x summary
==================
This test method tests ``assert.bitNumber.x.valueIsLessThan``
method of CNM_AssertionInterfaces library, 
it provides the possibility to handover test data via parameter 


.. <legal notes>

legal notes
=================
| SPDX-FileCopyrightText: © 2022 ekvip automation GmbH <info@ekvip.de>
| SPDX-License-Identifier: Apache-2.0
| For details check: Apache-2.0_

.. _Apache-2.0: https://www.apache.org/licenses/LICENSE-2.0

.. </legal notes>

parameters
==========

*)

METHOD testValueIsLessThan
VAR_INPUT
	(* for the test it's the parameter ``currentValue`` *)
	valueToTest	:__XWORD;
	(* for the test it's the parameter ``greaterValue`` *)
	greater		:__XWORD;
END_VAR
VAR
	(* just the expectation if the assertion to test must be worng or true *)
	assertionIsWrong		:BOOL;
	(* contains the format string for the test message *)
	message					:Tc2_System.T_MaxString;
	(* TwinCAT printf with the test message *)
	messageStringBuilder	:Tc2_Utilities.FB_FormatString;
END_VAR
THIS^.assertorContainer.resetAssertor();

assertionIsWrong := (valueToTest >= greater);
message := SEL(
	assertionIsWrong,
	'currentValue is %d greaterValue is %d assertion must be TRUE',
	'currentValue is %d greaterValue is %d assertion must be FALSE'
);
messageStringBuilder(
	sFormat := message,
	arg1 := THIS^.AnyToArg(valueToTest),
	arg2 := THIS^.AnyToArg(greater)
);

THIS^.assertorContainer.assertor.assert.bitNumber.x.valueIsLessThan(
	currentValue := valueToTest,
	greaterValue := greater,
	message := ''
);

THIS^.AssertEquals_BOOL(
	Expected 	:= assertionIsWrong,
	Actual 		:= THIS^.assertorContainer.wasAssertionWrong,
	Message 	:= messageStringBuilder.sOut
);
END_METHOD

(*

x summary
==================
This test method tests ``assert.bitNumber.x.valueIsMax``
method of CNM_AssertionInterfaces library, 
it provides the possibility to handover test data via parameter 


.. <legal notes>

legal notes
=================
| SPDX-FileCopyrightText: © 2022 ekvip automation GmbH <info@ekvip.de>
| SPDX-License-Identifier: Apache-2.0
| For details check: Apache-2.0_

.. _Apache-2.0: https://www.apache.org/licenses/LICENSE-2.0

.. </legal notes>

parameters
==========

*)

METHOD testValueIsMax 
VAR_INPUT
	(* for the test it's the parameter ``currentValue`` *)
	valueToTest	:__XWORD;
	(* for the test it's the parameter ``maximumValue`` *)
	maximum		:__XWORD;
END_VAR
VAR
	(* just the expectation if the assertion to test must be worng or true *)
	assertionIsWrong		:BOOL;
	(* contains the format string for the test message *)
	message					:Tc2_System.T_MaxString;
	(* TwinCAT printf with the test message *)
	messageStringBuilder	:Tc2_Utilities.FB_FormatString;
END_VAR
THIS^.assertorContainer.resetAssertor();

assertionIsWrong := (valueToTest > maximum);
message := SEL(
	assertionIsWrong,
	'currentValue is %d maximumValue is %d assertion must be TRUE',
	'currentValue is %d maximumValue is %d assertion must be FALSE'
);
messageStringBuilder(
	sFormat := message,
	arg1 := THIS^.AnyToArg(valueToTest),
	arg2 := THIS^.AnyToArg(maximum)
);

THIS^.assertorContainer.assertor.assert.bitNumber.x.valueIsMax(
	currentValue := valueToTest,
	maximumValue := maximum,
	message := ''
);

THIS^.AssertEquals_BOOL(
	Expected 	:= assertionIsWrong,
	Actual 		:= THIS^.assertorContainer.wasAssertionWrong,
	Message 	:= messageStringBuilder.sOut
);
END_METHOD

(*

x summary
==================
This test method tests ``assert.bitNumber.x.valueIsMin``
method of CNM_AssertionInterfaces library, 
it provides the possibility to handover test data via parameter 


.. <legal notes>

legal notes
=================
| SPDX-FileCopyrightText: © 2022 ekvip automation GmbH <info@ekvip.de>
| SPDX-License-Identifier: Apache-2.0
| For details check: Apache-2.0_

.. _Apache-2.0: https://www.apache.org/licenses/LICENSE-2.0

.. </legal notes>

parameters
==========

*)

METHOD testValueIsMin 
VAR_INPUT
	(* for the test it's the parameter ``currentValue`` *)
	valueToTest	:__XWORD;
	(* for the test it's the parameter ``minimumValue`` *)
	minimum		:__XWORD;
END_VAR
VAR
	(* just the expectation if the assertion to test must be worng or true *)
	assertionIsWrong		:BOOL;
	(* contains the format string for the test message *)
	message					:Tc2_System.T_MaxString;
	(* TwinCAT printf with the test message *)
	messageStringBuilder	:Tc2_Utilities.FB_FormatString;
END_VAR
THIS^.assertorContainer.resetAssertor();

assertionIsWrong := (valueToTest < minimum);
message := SEL(
	assertionIsWrong,
	'currentValue is %d minimumValue is %d assertion must be TRUE',
	'currentValue is %d minimumValue is %d assertion must be FALSE'
);
messageStringBuilder(
	sFormat := message,
	arg1 := THIS^.AnyToArg(valueToTest),
	arg2 := THIS^.AnyToArg(minimum)
);

THIS^.assertorContainer.assertor.assert.bitNumber.x.valueIsMin(
	currentValue := valueToTest,
	minimumValue := minimum,
	message := ''
);

THIS^.AssertEquals_BOOL(
	Expected 	:= assertionIsWrong,
	Actual 		:= THIS^.assertorContainer.wasAssertionWrong,
	Message 	:= messageStringBuilder.sOut
);
END_METHOD

(*

x summary
==================
This test method tests ``assert.bitNumber.x.valueIsNotEqualTo``
method of CNM_AssertionInterfaces library, 
it provides the possibility to handover test data via parameter 


.. <legal notes>

legal notes
=================
| SPDX-FileCopyrightText: © 2022 ekvip automation GmbH <info@ekvip.de>
| SPDX-License-Identifier: Apache-2.0
| For details check: Apache-2.0_

.. _Apache-2.0: https://www.apache.org/licenses/LICENSE-2.0

.. </legal notes>

parameters
==========

*)

METHOD testValueIsNotEqualTo
VAR_INPUT
	(* for the test it's the parameter ``currentValue`` *)
	valueToTest	:__XWORD;
	(* for the test it's the parameter ``unexpectedValue`` *)
	unexpected	:__XWORD;
END_VAR
VAR
	(* just the expectation if the assertion to test must be worng or true *)
	assertionIsWrong		:BOOL;
	(* contains the format string for the test message *)
	message					:Tc2_System.T_MaxString;
	(* TwinCAT printf with the test message *)
	messageStringBuilder	:Tc2_Utilities.FB_FormatString;
END_VAR
THIS^.assertorContainer.resetAssertor();

assertionIsWrong := (valueToTest = unexpected);
message := SEL(
	assertionIsWrong,
	'currentValue is %d unexpectedValue is %d assertion must be TRUE', 
	'currentValue is %d unexpectedValue is %d assertion must be FALSE'
);
messageStringBuilder(
	sFormat := message,
	arg1 := THIS^.AnyToArg(valueToTest),
	arg2 := THIS^.AnyToArg(unexpected)
);

THIS^.assertorContainer.assertor.assert.bitNumber.x.valueIsNotEqualTo(
	currentValue := valueToTest,
	unexpectedValue := unexpected,
	message := ''
);

THIS^.AssertEquals_BOOL(
	Expected 	:= assertionIsWrong,
	Actual 		:= THIS^.assertorContainer.wasAssertionWrong,
	Message 	:= messageStringBuilder.sOut
);
END_METHOD

(*

x summary
==================
This test method tests ``assert.bitNumber.x.xorMaskIsEqualTo``
method of CNM_AssertionInterfaces library, 
it provides the possibility to handover test data via parameter 


.. <legal notes>

legal notes
=================
| SPDX-FileCopyrightText: © 2022 ekvip automation GmbH <info@ekvip.de>
| SPDX-License-Identifier: Apache-2.0
| For details check: Apache-2.0_

.. _Apache-2.0: https://www.apache.org/licenses/LICENSE-2.0

.. </legal notes>

parameters
==========

*)

METHOD testXorMaskIsEqualTo 
VAR_INPUT
	(* for the test it's the parameter ``currentValue`` *)
	valueToTest	:__XWORD;
	(* it's the mask for the currentValue *)
	mask		:__XWORD;
	(* for the test it's the parameter ``expectedValue`` *)
	expected	:__XWORD;
END_VAR
VAR
	(* just the expectation if the assertion to test must be worng or true *)
	assertionIsWrong		:BOOL;
	(* result of the bit operation to determine the value of ``assertionIsWrong`` *)
	result					:__XWORD;
	(* contains the format string for the test message *)
	message					:Tc2_System.T_MaxString;
	(* TwinCAT printf with the test message *)
	messageStringBuilder	:Tc2_Utilities.FB_FormatString;
END_VAR
THIS^.assertorContainer.resetAssertor();

result := (valueToTest XOR mask);
assertionIsWrong := (result <> expected);
message := SEL(
	assertionIsWrong,
	'currentValue: 16#%.16X XOR mask: 16#%.16X is 16#%.16X expectedValue: 16#%.16X assertion must be TRUE', 
	'currentValue: 16#%.16X XOR mask: 16#%.16X is 16#%.16X expectedValue: 16#%.16X assertion must be FALSE'
);
messageStringBuilder(
	sFormat := message,
	arg1 := THIS^.AnyToArg(valueToTest),
	arg2 := THIS^.AnyToArg(mask),
	arg3 := THIS^.AnyToArg(result),
	arg4 := THIS^.AnyToArg(expected)
);

THIS^.assertorContainer.assertor.assert.bitNumber.x.xorMaskIsEqualTo(
	currentValue	:= valueToTest,
	mask 			:= mask,
	expectedValue	:= expected,
	message			:= ''
);

THIS^.AssertEquals_BOOL(
	Expected 	:= assertionIsWrong,
	Actual 		:= THIS^.assertorContainer.wasAssertionWrong,
	Message 	:= messageStringBuilder.sOut
);
END_METHOD

(*

x summary
==================
This test method tests ``assert.bitNumber.x.xorMaskIsNotEqualTo``
method of CNM_AssertionInterfaces library, 
it provides the possibility to handover test data via parameter 


.. <legal notes>

legal notes
=================
| SPDX-FileCopyrightText: © 2022 ekvip automation GmbH <info@ekvip.de>
| SPDX-License-Identifier: Apache-2.0
| For details check: Apache-2.0_

.. _Apache-2.0: https://www.apache.org/licenses/LICENSE-2.0

.. </legal notes>

parameters
==========

*)

METHOD testXorMaskIsNotEqualTo 
VAR_INPUT
	(* for the test it's the parameter ``currentValue`` *)
	valueToTest	:__XWORD;
	(* it's the mask for the currentValue *)
	mask		:__XWORD;
	(* for the test it's the parameter ``unexpectedValue`` *)
	unexpected	:__XWORD;
END_VAR
VAR
	(* just the expectation if the assertion to test must be worng or true *)
	assertionIsWrong		:BOOL;
	(* result of the bit operation to determine the value of ``assertionIsWrong`` *)
	result					:__XWORD;
	(* contains the format string for the test message *)
	message					:Tc2_System.T_MaxString;
	(* TwinCAT printf with the test message *)
	messageStringBuilder	:Tc2_Utilities.FB_FormatString;
END_VAR
THIS^.assertorContainer.resetAssertor();

result := (valueToTest XOR mask);
assertionIsWrong := (result = unexpected);
message := SEL(
	assertionIsWrong,
	'currentValue: 16#%.16X XOR mask: 16#%.16X is 16#%.16X unexpectedValue: 16#%.16X assertion must be TRUE', 
	'currentValue: 16#%.16X XOR mask: 16#%.16X is 16#%.16X unexpectedValue: 16#%.16X assertion must be FALSE'
);
messageStringBuilder(
	sFormat := message,
	arg1 := THIS^.AnyToArg(valueToTest),
	arg2 := THIS^.AnyToArg(mask),
	arg3 := THIS^.AnyToArg(result),
	arg4 := THIS^.AnyToArg(unexpected)
);

THIS^.assertorContainer.assertor.assert.bitNumber.x.xorMaskIsNotEqualTo(
	currentValue	:= valueToTest,
	mask 			:= mask,
	unexpectedValue	:= unexpected,
	message			:= ''
);

THIS^.AssertEquals_BOOL(
	Expected 	:= assertionIsWrong,
	Actual 		:= THIS^.assertorContainer.wasAssertionWrong,
	Message 	:= messageStringBuilder.sOut
);
END_METHOD

END_FUNCTION_BLOCK

// ---- AssertionTester/AssertionTests/BitNumberAssertions/classes/LWordAssertionTests.TcPOU
(*

long summary
==================
This class tests all methods of LWORD assertions
with various combinations of inputs and checks expected 
outputs are satisfied or not

.. <legal notes>

legal notes
=================
| SPDX-FileCopyrightText: © 2022 ekvip automation GmbH <info@ekvip.de>
| SPDX-License-Identifier: Apache-2.0
| For details check: Apache-2.0_

.. _Apache-2.0: https://www.apache.org/licenses/LICENSE-2.0

.. </legal notes>

methods and properties
======================

*)

FUNCTION_BLOCK LWordAssertionTests EXTENDS AbstractAssertorTest
VAR_INPUT
END_VAR
VAR CONSTANT
	(* number of the lsb *)
	FIRST_BIT				:USINT := 0;
	(* number of the msb *)
	LAST_BIT				:USINT := 63;
	(* just the value zero *)
	ZERO					:LINT := 0;
	(* no single bit is set, it's just the value zero *)
	NO_BIT_SET				:LWORD := 16#0000_0000_0000_0000;
	(* just the lsb is set, it's just the value one *)
	LSB_ONLY				:LWORD := 16#0000_0000_0000_0001;
	(* all bits are set *)
	ALL_BITS_SET			:LWORD := 16#FFFF_FFFF_FFFF_FFFF;
	(* the msb is set only *)
	MSB_ONLY				:LWORD := 16#8000_0000_0000_0000;
	(* prefix to unify the test names *)
	TEST_NAME_PREFIX		:STRING := 'assert.bitNumber.long.';
	(* number how many times the product will be rotated right *)
	NUMBER_OF_RORS			:ULINT := 1;
	(* multiplicand for the ``multiplier`` *)
	MULTIPLICAND			:ULINT := 16#1111_1111_1111_1111;
	(* first of all multipliers the test iterates *)
	FIRST_MULTIPLIER		:ULINT := 0;
	(* first of all multipliers the test iterates *)
	LAST_MULTIPLIER			:ULINT := 15;
	(* constant for the modulo operator to check if valueToTest is even (lsb is unset) or odd (lsb is set) *)
	DEVISOR_FOR_EVEN_ODD	:ULINT := 2;
END_VAR

THIS^.runAndMaskIsEqualToTests();
THIS^.runAndMaskIsNotEqualToTests();
THIS^.runBitXIsEqualToTests();
THIS^.runBitXIsNotEqualToTests();
THIS^.runBitXIsSetTests();
THIS^.runBitXIsUnsetTests();
THIS^.runLsbIsEqualToTests();
THIS^.runLsbIsNotEqualToTests();
THIS^.runLsbIsSetTests();
THIS^.runLsbIsUnsetTests();
THIS^.runMsbIsEqualToTests();
THIS^.runMsbIsNotEqualToTests();
THIS^.runMsbIsSetTests();
THIS^.runMsbIsUnsetTests();
THIS^.runOrMaskIsEqualToTests();
THIS^.runOrMaskIsNotEqualToTests();
THIS^.runValueIsMaxTests();
THIS^.runValueIsMinTests();
THIS^.runValueIsEqualToTests();
THIS^.runValueIsGreaterTests();
THIS^.runValueIsLessThanTests();
THIS^.runValueIsInRangeOfTests();
THIS^.runValueIsNotEqualToTests();
THIS^.runXorMaskIsEqualToTests();
THIS^.runXorMaskIsNotEqualToTests();

(*

long summary
==================
This test method is a helper function to create a unified test name

.. <legal notes>

legal notes
=================
| SPDX-FileCopyrightText: © 2022 ekvip automation GmbH <info@ekvip.de>
| SPDX-License-Identifier: Apache-2.0
| For details check: Apache-2.0_

.. _Apache-2.0: https://www.apache.org/licenses/LICENSE-2.0

.. </legal notes>

parameters
==========

*)

METHOD PROTECTED getTestNameFor :Tc2_System.T_MaxString
VAR_INPUT
	(* name of the method to test, to create a unified test name *)
	nameOfMethodToTest	:Tc2_System.T_MaxString;
END_VAR
getTestNameFor := Tc2_Standard.CONCAT(THIS^.TEST_NAME_PREFIX, nameOfMethodToTest);
END_METHOD

(*

long summary
==================
This test method tests ``assert.bitNumber.long.andMaskIsEqualTo``
method of CNM_AssertionInterfaces library with various inputs

.. <legal notes>

legal notes
=================
| SPDX-FileCopyrightText: © 2022 ekvip automation GmbH <info@ekvip.de>
| SPDX-License-Identifier: Apache-2.0
| For details check: Apache-2.0_

.. _Apache-2.0: https://www.apache.org/licenses/LICENSE-2.0

.. </legal notes>

*)

METHOD runAndMaskIsEqualToTests
VAR
	(* shift to iterate through the bit numbers *)
	shift				:ULINT;
	(* mask with the bit iteration *)
	mask				:LWORD;
END_VAR
RETURN (NOT TcUnit.TEST_ORDERED(THIS^.getTestNameFor('AndMaskIsEqualTo')));

FOR shift:= THIS^.FIRST_BIT TO THIS^.LAST_BIT DO
	mask := SHL(THIS^.LSB_ONLY, shift);
	THIS^.testAndMaskIsEqualTo(
		valueToTest := THIS^.ALL_BITS_SET,
		mask  := mask,
		expected := mask
	);
	THIS^.testAndMaskIsEqualTo(
		valueToTest := THIS^.ALL_BITS_SET,
		mask  := mask,
		expected := (NOT mask)
	);
	THIS^.testAndMaskIsEqualTo(
		valueToTest := mask,
		mask  := (NOT mask),
		expected := THIS^.NO_BIT_SET
	);
	THIS^.testAndMaskIsEqualTo(
		valueToTest := mask,
		mask  := (NOT mask),
		expected := (NOT mask)
	);	
	THIS^.testAndMaskIsEqualTo(
		valueToTest := mask,
		mask  := mask,
		expected := mask
	);	
END_FOR

THIS^.testAndMaskIsEqualTo(
	valueToTest := THIS^.NO_BIT_SET,
	mask  := THIS^.NO_BIT_SET,
	expected := THIS^.NO_BIT_SET
);
THIS^.testAndMaskIsEqualTo(
	valueToTest := THIS^.NO_BIT_SET,
	mask  := THIS^.NO_BIT_SET,
	expected := THIS^.LSB_ONLY
);

THIS^.testAndMaskIsEqualTo(
	valueToTest := THIS^.ALL_BITS_SET,
	mask  := THIS^.ALL_BITS_SET,
	expected := THIS^.ALL_BITS_SET
);
THIS^.testAndMaskIsEqualTo(
	valueToTest := THIS^.ALL_BITS_SET,
	mask  := THIS^.ALL_BITS_SET,
	expected := THIS^.NO_BIT_SET
);

TcUnit.TEST_FINISHED();
END_METHOD

(*

long summary
==================
This test method tests ``assert.bitNumber.long.andMaskIsNotEqualTo``
method of CNM_AssertionInterfaces library with various inputs

.. <legal notes>

legal notes
=================
| SPDX-FileCopyrightText: © 2022 ekvip automation GmbH <info@ekvip.de>
| SPDX-License-Identifier: Apache-2.0
| For details check: Apache-2.0_

.. _Apache-2.0: https://www.apache.org/licenses/LICENSE-2.0

.. </legal notes>

*)

METHOD runAndMaskIsNotEqualToTests
VAR
	(* shift to iterate through the bit numbers *)
	shift	:ULINT;
	(* mask with the bit iteration *)
	mask	:LWORD;
END_VAR
RETURN (NOT TcUnit.TEST_ORDERED(THIS^.getTestNameFor('AndMaskIsNotEqualTo')));

FOR shift:= THIS^.FIRST_BIT TO THIS^.LAST_BIT DO
	mask := SHL(THIS^.LSB_ONLY, shift);
	THIS^.testAndMaskIsNotEqualTo(
		valueToTest := THIS^.ALL_BITS_SET,
		mask  := mask,
		unexpected := (NOT mask)
	);
	THIS^.testAndMaskIsNotEqualTo(
		valueToTest := THIS^.ALL_BITS_SET,
		mask  := mask,
		unexpected := mask
	);
	THIS^.testAndMaskIsNotEqualTo(
		valueToTest := mask,
		mask  := (NOT mask),
		unexpected := (NOT mask)
	);	
	THIS^.testAndMaskIsNotEqualTo(
		valueToTest := mask,
		mask  := (NOT mask),
		unexpected := THIS^.NO_BIT_SET
	);
	THIS^.testAndMaskIsNotEqualTo(
		valueToTest := mask,
		mask  := mask,
		unexpected := mask
	);	
END_FOR

THIS^.testAndMaskIsNotEqualTo(
	valueToTest := THIS^.NO_BIT_SET,
	mask  := THIS^.NO_BIT_SET,
	unexpected := THIS^.LSB_ONLY
);
THIS^.testAndMaskIsNotEqualTo(
	valueToTest := THIS^.NO_BIT_SET,
	mask  := THIS^.NO_BIT_SET,
	unexpected := THIS^.NO_BIT_SET
);

THIS^.testAndMaskIsNotEqualTo(
	valueToTest := THIS^.ALL_BITS_SET,
	mask  := THIS^.ALL_BITS_SET,
	unexpected := THIS^.NO_BIT_SET
);
THIS^.testAndMaskIsNotEqualTo(
	valueToTest := THIS^.ALL_BITS_SET,
	mask  := THIS^.ALL_BITS_SET,
	unexpected := THIS^.ALL_BITS_SET
);

TcUnit.TEST_FINISHED();
END_METHOD

(*

long summary
==================
This test method tests ``assert.bitNumber.long.bitXIsEqualTo``
method of CNM_AssertionInterfaces library with various inputs

.. <legal notes>

legal notes
=================
| SPDX-FileCopyrightText: © 2022 ekvip automation GmbH <info@ekvip.de>
| SPDX-License-Identifier: Apache-2.0
| For details check: Apache-2.0_

.. _Apache-2.0: https://www.apache.org/licenses/LICENSE-2.0

.. </legal notes>

*)

METHOD runBitXIsEqualToTests
VAR
	(* this is the number of the bit to test *)
	bitNumberToTest	:CNM_AssertionInterfaces.BitNumberLWord;
	(* it's just part of the test data *)
	valueToTest		:LWORD;
END_VAR
RETURN (NOT TcUnit.TEST_ORDERED(THIS^.getTestNameFor('bitXIsEqualTo')));

FOR bitNumberToTest := THIS^.FIRST_BIT TO THIS^.LAST_BIT DO

	valueToTest := SHL(THIS^.LSB_ONLY,bitNumberToTest);
	THIS^.testBitXIsEqualTo(
		valueToTest			:=valueToTest,
		bitNumberToCheck	:=bitNumberToTest,
		bitIsSet			:=TRUE
	);
	THIS^.testBitXIsEqualTo(
		valueToTest			:=valueToTest,
		bitNumberToCheck	:=bitNumberToTest,
		bitIsSet			:=FALSE
	);

	valueToTest := (NOT valueToTest);
	THIS^.testBitXIsEqualTo(
		valueToTest			:=valueToTest,
		bitNumberToCheck	:=bitNumberToTest,
		bitIsSet			:=FALSE
	);
	THIS^.testBitXIsEqualTo(
		valueToTest			:=valueToTest,
		bitNumberToCheck	:=bitNumberToTest,
		bitIsSet			:=TRUE
	);	
END_FOR

TcUnit.TEST_FINISHED();
END_METHOD

(*

long summary
==================
This test method tests ``assert.bitNumber.long.bitXIsNotEqualTo``
method of CNM_AssertionInterfaces library with various inputs

.. <legal notes>

legal notes
=================
| SPDX-FileCopyrightText: © 2022 ekvip automation GmbH <info@ekvip.de>
| SPDX-License-Identifier: Apache-2.0
| For details check: Apache-2.0_

.. _Apache-2.0: https://www.apache.org/licenses/LICENSE-2.0

.. </legal notes>

*)

METHOD runBitXIsNotEqualToTests
VAR
	(* this is the number of the bit to test *)
	bitNumberToTest	:CNM_AssertionInterfaces.BitNumberLWord;
	(* it's just part of the test data *)
	valueToTest		:LWORD;
END_VAR
RETURN (NOT TcUnit.TEST_ORDERED(THIS^.getTestNameFor('bitXIsNotEqualTo')));

FOR bitNumberToTest := THIS^.FIRST_BIT TO THIS^.LAST_BIT DO
	valueToTest := SHL(THIS^.LSB_ONLY,bitNumberToTest);
	THIS^.testBitXIsNotEqualTo(
		valueToTest			:=valueToTest,
		bitNumberToCheck	:=bitNumberToTest,
		bitIsSet			:=TRUE
	);
	THIS^.testBitXIsNotEqualTo(
		valueToTest			:=valueToTest,
		bitNumberToCheck	:=bitNumberToTest,
		bitIsSet			:=FALSE
	);

	valueToTest := (NOT valueToTest);
	THIS^.testBitXIsNotEqualTo(
		valueToTest			:=valueToTest,
		bitNumberToCheck	:=bitNumberToTest,
		bitIsSet			:=TRUE
	);
	THIS^.testBitXIsNotEqualTo(
		valueToTest			:=valueToTest,
		bitNumberToCheck	:=bitNumberToTest,
		bitIsSet			:=FALSE
	);	
END_FOR

TcUnit.TEST_FINISHED();
END_METHOD

(*

long summary
==================
This test method tests ``assert.bitNumber.long.bitXIsSet`` 
of CNM_AssertionInterfaces library with various inputs

.. <legal notes>

legal notes
=================
| SPDX-FileCopyrightText: © 2022 ekvip automation GmbH <info@ekvip.de>
| SPDX-License-Identifier: Apache-2.0
| For details check: Apache-2.0_

.. _Apache-2.0: https://www.apache.org/licenses/LICENSE-2.0

.. </legal notes>

*)

METHOD runBitXIsSetTests
VAR
	(* this is the number of the bit to test *)
	bitNumberToTest	:CNM_AssertionInterfaces.BitNumberLWord;
	(* it's just part of the test data *)
	valueToTest		:LWORD;
END_VAR
RETURN (NOT TcUnit.TEST_ORDERED(THIS^.getTestNameFor('bitXIsSet')));

FOR bitNumberToTest := THIS^.FIRST_BIT TO THIS^.LAST_BIT DO
	valueToTest := SHL(THIS^.LSB_ONLY,bitNumberToTest);
	THIS^.testBitXIsSet(
		valueToTest := valueToTest,
		bitNumberToCheck := bitNumberToTest
	);
	THIS^.testBitXIsSet(
		valueToTest := (NOT valueToTest),
		bitNumberToCheck := bitNumberToTest
	);
	THIS^.testBitXIsSet(
		valueToTest := THIS^.NO_BIT_SET,
		bitNumberToCheck := bitNumberToTest
	);
	THIS^.testBitXIsSet(
		valueToTest := THIS^.ALL_BITS_SET,
		bitNumberToCheck := bitNumberToTest
	);
END_FOR

TcUnit.TEST_FINISHED();
END_METHOD

(*

long summary
==================
This test method tests ``assert.bitNumber.long.bitXIsUnset``
of CNM_AssertionInterfaces library with various inputs

.. <legal notes>

legal notes
=================
| SPDX-FileCopyrightText: © 2022 ekvip automation GmbH <info@ekvip.de>
| SPDX-License-Identifier: Apache-2.0
| For details check: Apache-2.0_

.. _Apache-2.0: https://www.apache.org/licenses/LICENSE-2.0

.. </legal notes>

*)

METHOD runBitXIsUnsetTests
VAR
	(* this is the number of the bit to test *)
	bitNumberToTest	:CNM_AssertionInterfaces.BitNumberLWord;
	(* it's just part of the test data *)
	valueToTest		:LWORD;
END_VAR
RETURN (NOT TcUnit.TEST_ORDERED(THIS^.getTestNameFor('bitXIsUnset')));

FOR bitNumberToTest := THIS^.FIRST_BIT TO THIS^.LAST_BIT DO
	valueToTest := SHL(THIS^.LSB_ONLY,bitNumberToTest);
	THIS^.testBitXIsUnset(
		valueToTest := valueToTest,
		bitNumberToCheck := bitNumberToTest
	);
	THIS^.testBitXIsUnset(
		valueToTest := (NOT valueToTest),
		bitNumberToCheck := bitNumberToTest
	);
	THIS^.testBitXIsUnset(
		valueToTest := THIS^.NO_BIT_SET,
		bitNumberToCheck := bitNumberToTest
	);
	THIS^.testBitXIsUnset(
		valueToTest :=THIS^.ALL_BITS_SET,
		bitNumberToCheck := bitNumberToTest
	);
END_FOR

TcUnit.TEST_FINISHED();
END_METHOD

(*

long summary
==================
This test method tests ``assert.bitNumber.long.lsbIsEqualTo``
method of CNM_AssertionInterfaces library with various inputs

.. <legal notes>

legal notes
=================
| SPDX-FileCopyrightText: © 2022 ekvip automation GmbH <info@ekvip.de>
| SPDX-License-Identifier: Apache-2.0
| For details check: Apache-2.0_

.. _Apache-2.0: https://www.apache.org/licenses/LICENSE-2.0

.. </legal notes>

*)

METHOD runLsbIsEqualToTests
VAR
	(* it's just part of the test data *)
	valueToTest	:LWORD;
	(* multiplier to get various bit patterns *)
	multiplier	:ULINT;
END_VAR
RETURN (NOT TcUnit.TEST_ORDERED(THIS^.getTestNameFor('lsbIsEqualTo')));

FOR multiplier := THIS^.FIRST_MULTIPLIER TO THIS^.LAST_MULTIPLIER DO
	valueToTest := (THIS^.MULTIPLICAND * multiplier);

	THIS^.testLsbIsEqualTo(
		valueToTest := valueToTest,
		expectedValue := TRUE
	);	
	THIS^.testLsbIsEqualTo(
		valueToTest := valueToTest,
		expectedValue := FALSE
	);

END_FOR

THIS^.testLsbIsEqualTo(
	valueToTest := THIS^.LSB_ONLY,
	expectedValue := TRUE
);	
THIS^.testLsbIsEqualTo(
	valueToTest := THIS^.LSB_ONLY,
	expectedValue := FALSE
);
THIS^.testLsbIsEqualTo(
	valueToTest := THIS^.MSB_ONLY,
	expectedValue := TRUE
);	
THIS^.testLsbIsEqualTo(
	valueToTest := THIS^.MSB_ONLY,
	expectedValue := FALSE
);

TcUnit.TEST_FINISHED();
END_METHOD

(*

long summary
==================
This test method tests ``assert.bitNumber.long.lsbIsNotEqualTo``
method of CNM_AssertionInterfaces library with various inputs

.. <legal notes>

legal notes
=================
| SPDX-FileCopyrightText: © 2022 ekvip automation GmbH <info@ekvip.de>
| SPDX-License-Identifier: Apache-2.0
| For details check: Apache-2.0_

.. _Apache-2.0: https://www.apache.org/licenses/LICENSE-2.0

.. </legal notes>

*)

METHOD runLsbIsNotEqualToTests
VAR
	(* it's just part of the test data *)
	valueToTest	:LWORD;
	(* multiplier to get various bit patterns *)
	multiplier	:ULINT;
END_VAR
RETURN (NOT TcUnit.TEST_ORDERED(THIS^.getTestNameFor('lsbIsNotEqualTo')));

FOR multiplier := THIS^.FIRST_MULTIPLIER TO THIS^.LAST_MULTIPLIER DO
	valueToTest := (THIS^.MULTIPLICAND * multiplier);

	THIS^.testLsbIsNotEqualTo(
		valueToTest := valueToTest,
		unexpectedValue := TRUE
	);	
	THIS^.testLsbIsNotEqualTo(
		valueToTest := valueToTest,
		unexpectedValue := FALSE
	);

END_FOR

THIS^.testLsbIsNotEqualTo(
	valueToTest := THIS^.LSB_ONLY,
	unexpectedValue := TRUE
);	
THIS^.testLsbIsNotEqualTo(
	valueToTest := THIS^.LSB_ONLY,
	unexpectedValue := FALSE
);
THIS^.testLsbIsNotEqualTo(
	valueToTest := THIS^.MSB_ONLY,
	unexpectedValue := TRUE
);	
THIS^.testLsbIsNotEqualTo(
	valueToTest := THIS^.MSB_ONLY,
	unexpectedValue := FALSE
);

TcUnit.TEST_FINISHED();
END_METHOD

(*

long summary
==================
This test method tests ``assert.bitNumber.long.lsbIsSet``
of CNM_AssertionInterfaces library with various inputs

.. <legal notes>

legal notes
=================
| SPDX-FileCopyrightText: © 2022 ekvip automation GmbH <info@ekvip.de>
| SPDX-License-Identifier: Apache-2.0
| For details check: Apache-2.0_

.. _Apache-2.0: https://www.apache.org/licenses/LICENSE-2.0

.. </legal notes>

*)

METHOD runLsbIsSetTests
VAR
	(* it's just part of the test data *)
	valueToTest	:LWORD;
	(* multiplier to get various bit patterns *)
	multiplier	:ULINT;
END_VAR
RETURN (NOT TcUnit.TEST_ORDERED(THIS^.getTestNameFor('lsbIsSet')));

FOR multiplier := THIS^.FIRST_MULTIPLIER TO THIS^.LAST_MULTIPLIER DO
	valueToTest := (THIS^.MULTIPLICAND * multiplier);
	THIS^.testLsbIsSet(
		valueToTest := valueToTest
	);
END_FOR

THIS^.testLsbIsSet(
	valueToTest := THIS^.MSB_ONLY
);	
THIS^.testLsbIsSet(
	valueToTest := THIS^.MSB_ONLY
);

TcUnit.TEST_FINISHED();
END_METHOD

(*

long summary
==================
This test method tests ``assert.bitNumber.long.lsbIsUnset``
of CNM_AssertionInterfaces library with various inputs

.. <legal notes>

legal notes
=================
| SPDX-FileCopyrightText: © 2022 ekvip automation GmbH <info@ekvip.de>
| SPDX-License-Identifier: Apache-2.0
| For details check: Apache-2.0_

.. _Apache-2.0: https://www.apache.org/licenses/LICENSE-2.0

.. </legal notes>

*)

METHOD runLsbIsUnsetTests
VAR
	(* it's just part of the test data *)
	valueToTest	:LWORD;
	(* multiplier to get various bit patterns *)
	multiplier	:ULINT;
END_VAR
RETURN (NOT TcUnit.TEST_ORDERED(THIS^.getTestNameFor('lsbIsUnset')));

FOR multiplier := THIS^.FIRST_MULTIPLIER TO THIS^.LAST_MULTIPLIER DO
	valueToTest := (THIS^.MULTIPLICAND * multiplier);
	THIS^.testLsbIsUnset(
		valueToTest := valueToTest
	);
END_FOR

THIS^.testLsbIsUnset(
	valueToTest := THIS^.LSB_ONLY
);	
THIS^.testLsbIsUnset(
	valueToTest := THIS^.MSB_ONLY
);

TcUnit.TEST_FINISHED();
END_METHOD

(*

long summary
==================
This test method tests ``assert.bitNumber.long.msbIsEqualTo``
method of CNM_AssertionInterfaces library with various inputs

.. <legal notes>

legal notes
=================
| SPDX-FileCopyrightText: © 2022 ekvip automation GmbH <info@ekvip.de>
| SPDX-License-Identifier: Apache-2.0
| For details check: Apache-2.0_

.. _Apache-2.0: https://www.apache.org/licenses/LICENSE-2.0

.. </legal notes>

*)

METHOD runMsbIsEqualToTests
VAR
	(* it's just part of the test data *)
	valueToTest	:LWORD;
	(* multiplier to get various bit patterns *)
	multiplier	:ULINT;
END_VAR
VAR CONSTANT
	(* number how many times the product will be rotated right *)
	NUMBER_OF_RORS :ULINT := 1;
	(* multiplicand for the ``multiplier`` *)
	MULTIPLICAND :ULINT := 17;
	(* first of all multipliers the test iterates *)
	FIRST_MULTIPLIER :ULINT := 0;
	(* first of all multipliers the test iterates *)
	LAST_MULTIPLIER :ULINT := 15;
END_VAR
RETURN (NOT TcUnit.TEST_ORDERED(THIS^.getTestNameFor('msbIsEqualTo')));

FOR multiplier := THIS^.FIRST_MULTIPLIER TO THIS^.LAST_MULTIPLIER DO
	valueToTest := ROR(THIS^.MULTIPLICAND * multiplier, THIS^.NUMBER_OF_RORS);

	THIS^.testMsbIsEqualTo(
		valueToTest := valueToTest,
		expectedValue := TRUE
	);	
	THIS^.testMsbIsEqualTo(
		valueToTest := valueToTest,
		expectedValue := FALSE
	);
END_FOR

THIS^.testMsbIsEqualTo(
	valueToTest := THIS^.LSB_ONLY,
	expectedValue := TRUE
);	
THIS^.testMsbIsEqualTo(
	valueToTest := THIS^.LSB_ONLY,
	expectedValue := FALSE
);
THIS^.testMsbIsEqualTo(
	valueToTest := THIS^.MSB_ONLY,
	expectedValue := TRUE
);	
THIS^.testMsbIsEqualTo(
	valueToTest := THIS^.MSB_ONLY,
	expectedValue := FALSE
);

TcUnit.TEST_FINISHED();
END_METHOD

(*

long summary
==================
This test method tests ``assert.bitNumber.long.msbIsNotEqualTo``
method of CNM_AssertionInterfaces library with various inputs

.. <legal notes>

legal notes
=================
| SPDX-FileCopyrightText: © 2022 ekvip automation GmbH <info@ekvip.de>
| SPDX-License-Identifier: Apache-2.0
| For details check: Apache-2.0_

.. _Apache-2.0: https://www.apache.org/licenses/LICENSE-2.0

.. </legal notes>

*)

METHOD runMsbIsNotEqualToTests
VAR
	(* it's just part of the test data *)
	valueToTest	:LWORD;
	(* multiplier to get various bit patterns *)
	multiplier	:ULINT;
END_VAR
RETURN (NOT TcUnit.TEST_ORDERED(THIS^.getTestNameFor('msbIsNotEqualTo')));

FOR multiplier := THIS^.FIRST_MULTIPLIER TO THIS^.LAST_MULTIPLIER DO
	valueToTest := ROR(THIS^.MULTIPLICAND * multiplier, THIS^.NUMBER_OF_RORS);
	THIS^.testMsbIsNotEqualTo(
		valueToTest := valueToTest,
		unexpectedValue := TRUE
	);	
	THIS^.testMsbIsNotEqualTo(
		valueToTest := valueToTest,
		unexpectedValue := FALSE
	);
END_FOR

THIS^.testMsbIsNotEqualTo(
	valueToTest := THIS^.LSB_ONLY,
	unexpectedValue := TRUE
);	
THIS^.testMsbIsNotEqualTo(
	valueToTest := THIS^.LSB_ONLY,
	unexpectedValue := FALSE
);
THIS^.testMsbIsNotEqualTo(
	valueToTest := THIS^.MSB_ONLY,
	unexpectedValue := TRUE
);	
THIS^.testMsbIsNotEqualTo(
	valueToTest := THIS^.MSB_ONLY,
	unexpectedValue := FALSE
);

TcUnit.TEST_FINISHED();
END_METHOD

(*

long summary
==================
This test method tests ``assert.bitNumber.long.msbIsSet``
of CNM_AssertionInterfaces library with various inputs

.. <legal notes>

legal notes
=================
| SPDX-FileCopyrightText: © 2022 ekvip automation GmbH <info@ekvip.de>
| SPDX-License-Identifier: Apache-2.0
| For details check: Apache-2.0_

.. _Apache-2.0: https://www.apache.org/licenses/LICENSE-2.0

.. </legal notes>

*)

METHOD runMsbIsSetTests
VAR
	(* it's just part of the test data *)
	valueToTest	:LWORD;
	(* multiplier to get various bit patterns *)
	multiplier	:ULINT;
END_VAR
RETURN (NOT TcUnit.TEST_ORDERED(THIS^.getTestNameFor('msbIsUnset')));

FOR multiplier := THIS^.FIRST_MULTIPLIER TO THIS^.LAST_MULTIPLIER DO
	valueToTest := ROR(THIS^.MULTIPLICAND * multiplier, THIS^.NUMBER_OF_RORS);
	THIS^.testMsbIsSet(
		valueToTest := valueToTest
	);
END_FOR

THIS^.testMsbIsSet(
	valueToTest := THIS^.LSB_ONLY
);	
THIS^.testMsbIsSet(
	valueToTest := THIS^.MSB_ONLY
);

TcUnit.TEST_FINISHED();
END_METHOD

(*

long summary
==================
This test method tests ``assert.bitNumber.long.msbIsUnset``
of CNM_AssertionInterfaces library with various inputs

.. <legal notes>

legal notes
=================
| SPDX-FileCopyrightText: © 2022 ekvip automation GmbH <info@ekvip.de>
| SPDX-License-Identifier: Apache-2.0
| For details check: Apache-2.0_

.. _Apache-2.0: https://www.apache.org/licenses/LICENSE-2.0

.. </legal notes>

*)

METHOD runMsbIsUnsetTests
VAR
	(* it's just part of the test data *)
	valueToTest	:LWORD;
	(* multiplier to get various bit patterns *)
	multiplier	:ULINT;
END_VAR
RETURN (NOT TcUnit.TEST_ORDERED(THIS^.getTestNameFor('msbIsSet')));

FOR multiplier := THIS^.FIRST_MULTIPLIER TO THIS^.LAST_MULTIPLIER DO
	valueToTest := ROR(THIS^.MULTIPLICAND * multiplier, THIS^.NUMBER_OF_RORS);
	THIS^.testMsbIsSet(
		valueToTest := valueToTest
	);
END_FOR

THIS^.testMsbIsSet(
	valueToTest := THIS^.LSB_ONLY
);	
THIS^.testMsbIsSet(
	valueToTest := THIS^.MSB_ONLY
);

TcUnit.TEST_FINISHED();
END_METHOD

(*

long summary
==================
This test method tests ``assert.bitNumber.long.orMaskIsEqualTo``
method of CNM_AssertionInterfaces library with various inputs

.. <legal notes>

legal notes
=================
| SPDX-FileCopyrightText: © 2022 ekvip automation GmbH <info@ekvip.de>
| SPDX-License-Identifier: Apache-2.0
| For details check: Apache-2.0_

.. _Apache-2.0: https://www.apache.org/licenses/LICENSE-2.0

.. </legal notes>

*)

METHOD runOrMaskIsEqualToTests
VAR
	(* shift to iterate through the bit numbers *)
	shift				:ULINT;
	(* it's just part of the test data *)
	valueToTest		:LWORD;
	(* mask with the bit iteration *)
	mask				:LWORD;
END_VAR
RETURN (NOT TcUnit.TEST_ORDERED(THIS^.getTestNameFor('orMaskIsEqualTo')));

FOR shift:= THIS^.FIRST_BIT TO THIS^.LAST_BIT DO
	mask := SHL(THIS^.LSB_ONLY, shift);
	valueToTest := SHR(THIS^.MSB_ONLY, shift);
	THIS^.testOrMaskIsEqualTo(
		valueToTest := valueToTest,
		mask  := mask,
		expected := (mask OR valueToTest)
	);
	THIS^.testOrMaskIsEqualTo(
		valueToTest := valueToTest,
		mask  := mask,
		expected := (NOT (mask OR valueToTest))
	);
	THIS^.testAndMaskIsEqualTo(
		valueToTest := mask,
		mask  := (NOT mask),
		expected := THIS^.NO_BIT_SET
	);
	THIS^.testAndMaskIsEqualTo(
		valueToTest := mask,
		mask  := (NOT mask),
		expected := THIS^.ALL_BITS_SET
	);	
END_FOR

THIS^.testAndMaskIsEqualTo(
	valueToTest := THIS^.NO_BIT_SET,
	mask  := THIS^.NO_BIT_SET,
	expected := THIS^.NO_BIT_SET
);
THIS^.testAndMaskIsEqualTo(
	valueToTest := THIS^.NO_BIT_SET,
	mask  := THIS^.NO_BIT_SET,
	expected := THIS^.ALL_BITS_SET
);	

THIS^.testAndMaskIsEqualTo(
	valueToTest := THIS^.ALL_BITS_SET,
	mask  := THIS^.ALL_BITS_SET,
	expected := THIS^.ALL_BITS_SET
);
THIS^.testAndMaskIsEqualTo(
	valueToTest := THIS^.ALL_BITS_SET,
	mask  := THIS^.ALL_BITS_SET,
	expected := THIS^.NO_BIT_SET
);	

TcUnit.TEST_FINISHED();
END_METHOD

(*

long summary
==================
This test method tests ``assert.bitNumber.long.orMaskIsNotEqualTo``
method of CNM_AssertionInterfaces library with various inputs

.. <legal notes>

legal notes
=================
| SPDX-FileCopyrightText: © 2022 ekvip automation GmbH <info@ekvip.de>
| SPDX-License-Identifier: Apache-2.0
| For details check: Apache-2.0_

.. _Apache-2.0: https://www.apache.org/licenses/LICENSE-2.0

.. </legal notes>

*)

METHOD runOrMaskIsNotEqualToTests
VAR
	(* shift to iterate through the bit numbers *)
	shift				:ULINT;
	(* it's just part of the test data *)
	valueToTest		:LWORD;
	(* mask with the bit iteration *)
	mask				:LWORD;
END_VAR
RETURN (NOT TcUnit.TEST_ORDERED(THIS^.getTestNameFor('orMaskIsNotEqualTo')));

FOR shift:= THIS^.FIRST_BIT TO THIS^.LAST_BIT DO
	mask := SHL(THIS^.LSB_ONLY, shift);
	valueToTest := SHR(THIS^.MSB_ONLY, shift);
	THIS^.testOrMaskIsNotEqualTo(
		valueToTest := valueToTest,
		mask  := mask,
		unexpected := (mask OR valueToTest)
	);
	THIS^.testOrMaskIsNotEqualTo(
		valueToTest := valueToTest,
		mask  := mask,
		unexpected := (NOT (mask OR valueToTest))
	);
	THIS^.testOrMaskIsNotEqualTo(
		valueToTest := mask,
		mask  := (NOT mask),
		unexpected := THIS^.NO_BIT_SET
	);
	THIS^.testOrMaskIsNotEqualTo(
		valueToTest := mask,
		mask  := (NOT mask),
		unexpected := THIS^.ALL_BITS_SET
	);	
END_FOR

THIS^.testOrMaskIsNotEqualTo(
	valueToTest := THIS^.NO_BIT_SET,
	mask  := THIS^.NO_BIT_SET,
	unexpected := THIS^.NO_BIT_SET
);
THIS^.testOrMaskIsNotEqualTo(
	valueToTest := THIS^.NO_BIT_SET,
	mask  := THIS^.NO_BIT_SET,
	unexpected := THIS^.ALL_BITS_SET
);	

THIS^.testOrMaskIsNotEqualTo(
	valueToTest := THIS^.ALL_BITS_SET,
	mask  := THIS^.ALL_BITS_SET,
	unexpected := THIS^.ALL_BITS_SET
);
THIS^.testOrMaskIsNotEqualTo(
	valueToTest := THIS^.ALL_BITS_SET,
	mask  := THIS^.ALL_BITS_SET,
	unexpected := THIS^.NO_BIT_SET
);	

TcUnit.TEST_FINISHED();
END_METHOD

(*

long summary
==================
This test method tests ``assert.bitNumber.long.valueIsEqualTo``
method of CNM_AssertionInterfaces library with various inputs

.. <legal notes>

legal notes
=================
| SPDX-FileCopyrightText: © 2022 ekvip automation GmbH <info@ekvip.de>
| SPDX-License-Identifier: Apache-2.0
| For details check: Apache-2.0_

.. _Apache-2.0: https://www.apache.org/licenses/LICENSE-2.0

.. </legal notes>

*)

METHOD runValueIsEqualToTests
RETURN (NOT TcUnit.TEST_ORDERED(THIS^.getTestNameFor('valueIsEqualTo')));

THIS^.testValueIsEqualTo(
	valueToTest := THIS^.NO_BIT_SET,
	expected := THIS^.ALL_BITS_SET
);
THIS^.testValueIsEqualTo(
	valueToTest := THIS^.NO_BIT_SET,
	expected := THIS^.NO_BIT_SET
);
THIS^.testValueIsEqualTo(
	valueToTest := THIS^.ALL_BITS_SET,
	expected := THIS^.ALL_BITS_SET
);
THIS^.testValueIsEqualTo(
	valueToTest := THIS^.ALL_BITS_SET,
	expected := THIS^.NO_BIT_SET
);
THIS^.testValueIsEqualTo(
	valueToTest := THIS^.LSB_ONLY,
	expected := THIS^.LSB_ONLY
);
THIS^.testValueIsEqualTo(
	valueToTest := THIS^.LSB_ONLY,
	expected := THIS^.MSB_ONLY
);
THIS^.testValueIsEqualTo(
	valueToTest := THIS^.MSB_ONLY,
	expected := THIS^.MSB_ONLY
);
THIS^.testValueIsEqualTo(
	valueToTest := THIS^.MSB_ONLY,
	expected := THIS^.LSB_ONLY
);

TcUnit.TEST_FINISHED();
END_METHOD

(*

long summary
==================
This test method tests ``assert.bitNumber.long.valueIsGreaterThan``
method of CNM_AssertionInterfaces library with various inputs

.. <legal notes>

legal notes
=================
| SPDX-FileCopyrightText: © 2022 ekvip automation GmbH <info@ekvip.de>
| SPDX-License-Identifier: Apache-2.0
| For details check: Apache-2.0_

.. _Apache-2.0: https://www.apache.org/licenses/LICENSE-2.0

.. </legal notes>

*)

METHOD runValueIsGreaterTests
RETURN (NOT TcUnit.TEST_ORDERED(THIS^.getTestNameFor('valueIsGreaterThan')));

THIS^.testValueIsGreater(
	valueToTest := THIS^.NO_BIT_SET,
	less := THIS^.ALL_BITS_SET
);
THIS^.testValueIsGreater(
	valueToTest := THIS^.NO_BIT_SET,
	less := THIS^.NO_BIT_SET
);
THIS^.testValueIsGreater(
	valueToTest := THIS^.ALL_BITS_SET,
	less := THIS^.ALL_BITS_SET
);
THIS^.testValueIsGreater(
	valueToTest := THIS^.ALL_BITS_SET,
	less := THIS^.NO_BIT_SET
);
THIS^.testValueIsGreater(
	valueToTest := THIS^.LSB_ONLY,
	less := THIS^.LSB_ONLY
);
THIS^.testValueIsGreater(
	valueToTest := THIS^.LSB_ONLY,
	less := THIS^.NO_BIT_SET
);
THIS^.testValueIsGreater(
	valueToTest := THIS^.LSB_ONLY,
	less := (THIS^.LSB_ONLY+THIS^.LSB_ONLY)
);
THIS^.testValueIsGreater(
	valueToTest := THIS^.MSB_ONLY,
	less := THIS^.MSB_ONLY
);
THIS^.testValueIsGreater(
	valueToTest := THIS^.MSB_ONLY,
	less := (NOT THIS^.MSB_ONLY)
);
THIS^.testValueIsGreater(
	valueToTest := THIS^.MSB_ONLY,
	less := THIS^.ALL_BITS_SET
);

TcUnit.TEST_FINISHED();
END_METHOD

(*

long summary
==================
This test method tests ``assert.bitNumber.long.valueIsInRangeOf``
method of CNM_AssertionInterfaces library with various inputs

.. <legal notes>

legal notes
=================
| SPDX-FileCopyrightText: © 2022 ekvip automation GmbH <info@ekvip.de>
| SPDX-License-Identifier: Apache-2.0
| For details check: Apache-2.0_

.. _Apache-2.0: https://www.apache.org/licenses/LICENSE-2.0

.. </legal notes>

*)

METHOD runValueIsInRangeOfTests
RETURN (NOT TcUnit.TEST_ORDERED(THIS^.getTestNameFor('valueIsInRangeOf')));

THIS^.testValueIsInRangeOf(
	lower := THIS^.NO_BIT_SET,
	valueToTest := THIS^.LSB_ONLY,
	upper := THIS^.ALL_BITS_SET
);
THIS^.testValueIsInRangeOf(
	lower := THIS^.NO_BIT_SET,
	valueToTest := THIS^.NO_BIT_SET,
	upper := THIS^.NO_BIT_SET
);
THIS^.testValueIsInRangeOf(
	lower := THIS^.ALL_BITS_SET,
	valueToTest := THIS^.ALL_BITS_SET,
	upper := THIS^.ALL_BITS_SET
);
THIS^.testValueIsInRangeOf(
	lower := THIS^.ALL_BITS_SET,
	valueToTest := THIS^.LSB_ONLY,
	upper := THIS^.NO_BIT_SET
);
THIS^.testValueIsInRangeOf(
	lower := THIS^.ALL_BITS_SET,
	valueToTest := THIS^.NO_BIT_SET,
	upper := THIS^.NO_BIT_SET
);

TEST_FINISHED();
END_METHOD

(*

long summary
==================
This test method tests ``assert.bitNumber.long.valueIsLessThan``
method of CNM_AssertionInterfaces library with various inputs

.. <legal notes>

legal notes
=================
| SPDX-FileCopyrightText: © 2022 ekvip automation GmbH <info@ekvip.de>
| SPDX-License-Identifier: Apache-2.0
| For details check: Apache-2.0_

.. _Apache-2.0: https://www.apache.org/licenses/LICENSE-2.0

.. </legal notes>

*)

METHOD runValueIsLessThanTests
RETURN (NOT TcUnit.TEST_ORDERED(THIS^.getTestNameFor('valueIsLessThan')));

THIS^.testValueIsLessThan(
	valueToTest := THIS^.NO_BIT_SET,
	greater := THIS^.ALL_BITS_SET
);
THIS^.testValueIsLessThan(
	valueToTest := THIS^.NO_BIT_SET,
	greater := THIS^.NO_BIT_SET
);
THIS^.testValueIsLessThan(
	valueToTest := THIS^.ALL_BITS_SET,
	greater := THIS^.ALL_BITS_SET
);
THIS^.testValueIsLessThan(
	valueToTest := THIS^.ALL_BITS_SET,
	greater := THIS^.NO_BIT_SET
);
THIS^.testValueIsLessThan(
	valueToTest := THIS^.LSB_ONLY,
	greater := THIS^.LSB_ONLY
);
THIS^.testValueIsLessThan(
	valueToTest := THIS^.LSB_ONLY,
	greater := THIS^.NO_BIT_SET
);
THIS^.testValueIsLessThan(
	valueToTest := THIS^.MSB_ONLY,
	greater := (THIS^.MSB_ONLY+THIS^.LSB_ONLY)
);
THIS^.testValueIsLessThan(
	valueToTest := THIS^.MSB_ONLY,
	greater := THIS^.MSB_ONLY
);
THIS^.testValueIsLessThan(
	valueToTest := THIS^.MSB_ONLY,
	greater := (NOT THIS^.MSB_ONLY)
);
THIS^.testValueIsLessThan(
	valueToTest := THIS^.MSB_ONLY,
	greater := THIS^.ALL_BITS_SET
);

TcUnit.TEST_FINISHED();
END_METHOD

(*

long summary
==================
This test method tests ``assert.bitNumber.long.valueIsMax``
method of CNM_AssertionInterfaces library with various inputs

.. <legal notes>

legal notes
=================
| SPDX-FileCopyrightText: © 2022 ekvip automation GmbH <info@ekvip.de>
| SPDX-License-Identifier: Apache-2.0
| For details check: Apache-2.0_

.. _Apache-2.0: https://www.apache.org/licenses/LICENSE-2.0

.. </legal notes>

*)

METHOD runValueIsMaxTests
RETURN (NOT TcUnit.TEST_ORDERED(THIS^.getTestNameFor('valueIsMax')));

THIS^.testValueIsMax(
	valueToTest := THIS^.NO_BIT_SET,
	maximum := THIS^.LSB_ONLY
);
THIS^.testValueIsMax(
	valueToTest := THIS^.LSB_ONLY,
	maximum := THIS^.NO_BIT_SET
);
THIS^.testValueIsMax(
	valueToTest := THIS^.NO_BIT_SET,
	maximum := THIS^.NO_BIT_SET
);
THIS^.testValueIsMax(
	valueToTest := THIS^.ALL_BITS_SET,
	maximum := ALL_BITS_SET
);
THIS^.testValueIsMax(
	valueToTest := (THIS^.ALL_BITS_SET-THIS^.LSB_ONLY),
	maximum := THIS^.ALL_BITS_SET
);
THIS^.testValueIsMax(
	valueToTest := THIS^.ALL_BITS_SET,
	maximum := (THIS^.ALL_BITS_SET-THIS^.LSB_ONLY)
);
THIS^.testValueIsMax(
	valueToTest := THIS^.MSB_ONLY,
	maximum := (THIS^.MSB_ONLY+THIS^.LSB_ONLY)
);
THIS^.testValueIsMax(
	valueToTest := (THIS^.MSB_ONLY+THIS^.LSB_ONLY),
	maximum := THIS^.MSB_ONLY
);
THIS^.testValueIsMax(
	valueToTest := THIS^.MSB_ONLY,
	maximum := (NOT THIS^.MSB_ONLY)
);
THIS^.testValueIsMax(
	valueToTest := (NOT THIS^.MSB_ONLY),
	maximum := THIS^.MSB_ONLY
);
THIS^.testValueIsMax(
	valueToTest := THIS^.MSB_ONLY,
	maximum := THIS^.MSB_ONLY
);

TcUnit.TEST_FINISHED();
END_METHOD

(*

long summary
==================
This test method tests ``assert.bitNumber.long.valueIsMin``
method of CNM_AssertionInterfaces library with various inputs

.. <legal notes>

legal notes
=================
| SPDX-FileCopyrightText: © 2022 ekvip automation GmbH <info@ekvip.de>
| SPDX-License-Identifier: Apache-2.0
| For details check: Apache-2.0_

.. _Apache-2.0: https://www.apache.org/licenses/LICENSE-2.0

.. </legal notes>

*)

METHOD runValueIsMinTests
RETURN (NOT TcUnit.TEST_ORDERED(THIS^.getTestNameFor('valueIsMin')));

THIS^.testValueIsMin(
	valueToTest := THIS^.NO_BIT_SET,
	minimum := THIS^.LSB_ONLY
);
THIS^.testValueIsMin(
	valueToTest := THIS^.LSB_ONLY,
	minimum := THIS^.NO_BIT_SET
);
THIS^.testValueIsMin(
	valueToTest := THIS^.NO_BIT_SET,
	minimum := THIS^.NO_BIT_SET
);
THIS^.testValueIsMin(
	valueToTest := THIS^.ALL_BITS_SET,
	minimum := ALL_BITS_SET
);
THIS^.testValueIsMin(
	valueToTest := (THIS^.ALL_BITS_SET-THIS^.LSB_ONLY),
	minimum := THIS^.ALL_BITS_SET
);
THIS^.testValueIsMin(
	valueToTest := THIS^.ALL_BITS_SET,
	minimum := (THIS^.ALL_BITS_SET-THIS^.LSB_ONLY)
);
THIS^.testValueIsMin(
	valueToTest := THIS^.MSB_ONLY,
	minimum := (THIS^.MSB_ONLY+THIS^.LSB_ONLY)
);
THIS^.testValueIsMin(
	valueToTest := (THIS^.MSB_ONLY+THIS^.LSB_ONLY),
	minimum := THIS^.MSB_ONLY
);
THIS^.testValueIsMin(
	valueToTest := THIS^.MSB_ONLY,
	minimum := (NOT THIS^.MSB_ONLY)
);
THIS^.testValueIsMin(
	valueToTest := (NOT THIS^.MSB_ONLY),
	minimum := THIS^.MSB_ONLY
);
THIS^.testValueIsMin(
	valueToTest := THIS^.MSB_ONLY,
	minimum := THIS^.MSB_ONLY
);

TcUnit.TEST_FINISHED();
END_METHOD

(*

long summary
==================
This test method tests ``assert.bitNumber.long.valueIsNotEqualTo``
method of CNM_AssertionInterfaces library with various inputs

.. <legal notes>

legal notes
=================
| SPDX-FileCopyrightText: © 2022 ekvip automation GmbH <info@ekvip.de>
| SPDX-License-Identifier: Apache-2.0
| For details check: Apache-2.0_

.. _Apache-2.0: https://www.apache.org/licenses/LICENSE-2.0

.. </legal notes>

*)

METHOD runValueIsNotEqualToTests
RETURN (NOT TcUnit.TEST_ORDERED(THIS^.getTestNameFor('valueIsNotEqualTo')));

THIS^.testValueIsNotEqualTo(
	valueToTest := THIS^.NO_BIT_SET,
	unexpected := THIS^.ALL_BITS_SET
);
THIS^.testValueIsNotEqualTo(
	valueToTest := THIS^.NO_BIT_SET,
	unexpected := THIS^.NO_BIT_SET
);
THIS^.testValueIsNotEqualTo(
	valueToTest := THIS^.ALL_BITS_SET,
	unexpected := THIS^.ALL_BITS_SET
);
THIS^.testValueIsNotEqualTo(
	valueToTest := THIS^.ALL_BITS_SET,
	unexpected := THIS^.NO_BIT_SET
);
THIS^.testValueIsNotEqualTo(
	valueToTest := THIS^.LSB_ONLY,
	unexpected := THIS^.LSB_ONLY
);
THIS^.testValueIsNotEqualTo(
	valueToTest := THIS^.LSB_ONLY,
	unexpected := THIS^.MSB_ONLY
);
THIS^.testValueIsNotEqualTo(
	valueToTest := THIS^.MSB_ONLY,
	unexpected := THIS^.MSB_ONLY
);
THIS^.testValueIsNotEqualTo(
	valueToTest := THIS^.MSB_ONLY,
	unexpected := THIS^.LSB_ONLY
);

TcUnit.TEST_FINISHED();
END_METHOD

(*

long summary
==================
This test method tests ``assert.bitNumber.long.xorMaskIsEqualTo``
method of CNM_AssertionInterfaces library with various inputs

.. <legal notes>

legal notes
=================
| SPDX-FileCopyrightText: © 2022 ekvip automation GmbH <info@ekvip.de>
| SPDX-License-Identifier: Apache-2.0
| For details check: Apache-2.0_

.. _Apache-2.0: https://www.apache.org/licenses/LICENSE-2.0

.. </legal notes>

*)

METHOD runXorMaskIsEqualToTests
VAR
	(* shift to iterate through the bit numbers *)
	shift				:ULINT;
	(* it's just part of the test data *)
	valueToTest		:LWORD;
	(* mask with the bit iteration *)
	mask				:LWORD;
END_VAR
RETURN (NOT TcUnit.TEST_ORDERED(THIS^.getTestNameFor('xorMaskIsEqualTo')));

FOR shift:= THIS^.FIRST_BIT TO THIS^.LAST_BIT DO
	mask := SHL(THIS^.LSB_ONLY, shift);
	valueToTest := (NOT mask);
	THIS^.testOrMaskIsEqualTo(
		valueToTest := valueToTest,
		mask  := mask,
		expected := THIS^.ALL_BITS_SET
	);
	THIS^.testOrMaskIsEqualTo(
		valueToTest := valueToTest,
		mask  := mask,
		expected := THIS^.NO_BIT_SET
	);
	THIS^.testAndMaskIsEqualTo(
		valueToTest := mask,
		mask  := mask,
		expected := THIS^.NO_BIT_SET
	);
	THIS^.testAndMaskIsEqualTo(
		valueToTest := mask,
		mask  := mask,
		expected := mask
	);	
END_FOR

THIS^.testAndMaskIsEqualTo(
	valueToTest := THIS^.NO_BIT_SET,
	mask  := THIS^.NO_BIT_SET,
	expected := THIS^.NO_BIT_SET
);
THIS^.testAndMaskIsEqualTo(
	valueToTest := THIS^.NO_BIT_SET,
	mask  := THIS^.NO_BIT_SET,
	expected := THIS^.ALL_BITS_SET
);	

THIS^.testAndMaskIsEqualTo(
	valueToTest := THIS^.ALL_BITS_SET,
	mask  := THIS^.ALL_BITS_SET,
	expected := THIS^.ALL_BITS_SET
);
THIS^.testAndMaskIsEqualTo(
	valueToTest := THIS^.ALL_BITS_SET,
	mask  := THIS^.ALL_BITS_SET,
	expected := THIS^.NO_BIT_SET
);	

TcUnit.TEST_FINISHED();
END_METHOD

(*

long summary
==================
This test method tests ``assert.bitNumber.long.xorMaskIsNotEqualTo``
method of CNM_AssertionInterfaces library with various inputs

.. <legal notes>

legal notes
=================
| SPDX-FileCopyrightText: © 2022 ekvip automation GmbH <info@ekvip.de>
| SPDX-License-Identifier: Apache-2.0
| For details check: Apache-2.0_

.. _Apache-2.0: https://www.apache.org/licenses/LICENSE-2.0

.. </legal notes>

*)

METHOD runXorMaskIsNotEqualToTests
VAR
	(* shift to iterate through the bit numbers *)
	shift				:ULINT;
	(* it's just part of the test data *)
	valueToTest			:LWORD;
	(* mask with the bit iteration *)
	mask				:LWORD;
END_VAR
RETURN (NOT TcUnit.TEST_ORDERED(THIS^.getTestNameFor('xorMaskIsNotEqualTo')));

FOR shift:= THIS^.FIRST_BIT TO THIS^.LAST_BIT DO
	mask := SHL(THIS^.LSB_ONLY, shift);
	valueToTest := (NOT mask);
	THIS^.testXorMaskIsNotEqualTo(
		valueToTest := valueToTest,
		mask  := mask,
		unexpected := THIS^.ALL_BITS_SET
	);
	THIS^.testXorMaskIsNotEqualTo(
		valueToTest := valueToTest,
		mask  := mask,
		unexpected := THIS^.NO_BIT_SET
	);
	THIS^.testXorMaskIsNotEqualTo(
		valueToTest := mask,
		mask  := mask,
		unexpected := THIS^.NO_BIT_SET
	);
	THIS^.testXorMaskIsNotEqualTo(
		valueToTest := mask,
		mask  := mask,
		unexpected := mask
	);	
END_FOR

THIS^.testXorMaskIsNotEqualTo(
	valueToTest := THIS^.NO_BIT_SET,
	mask  := THIS^.NO_BIT_SET,
	unexpected := THIS^.NO_BIT_SET
);
THIS^.testXorMaskIsNotEqualTo(
	valueToTest := THIS^.NO_BIT_SET,
	mask  := THIS^.NO_BIT_SET,
	unexpected := THIS^.ALL_BITS_SET
);	

THIS^.testXorMaskIsNotEqualTo(
	valueToTest := THIS^.ALL_BITS_SET,
	mask  := THIS^.ALL_BITS_SET,
	unexpected := THIS^.ALL_BITS_SET
);
THIS^.testXorMaskIsNotEqualTo(
	valueToTest := THIS^.ALL_BITS_SET,
	mask  := THIS^.ALL_BITS_SET,
	unexpected := THIS^.NO_BIT_SET
);	

THIS^.testXorMaskIsNotEqualTo(
	valueToTest := THIS^.ALL_BITS_SET,
	mask  := THIS^.NO_BIT_SET,
	unexpected := THIS^.ALL_BITS_SET
);
THIS^.testXorMaskIsNotEqualTo(
	valueToTest := THIS^.ALL_BITS_SET,
	mask  := THIS^.NO_BIT_SET,
	unexpected := THIS^.NO_BIT_SET
);

TcUnit.TEST_FINISHED();
END_METHOD

(*

long summary
==================
This test method tests ``assert.bitNumber.long.andMaskIsEqualTo``
method of CNM_AssertionInterfaces library, 
it provides the possibility to handover test data via parameter 


.. <legal notes>

legal notes
=================
| SPDX-FileCopyrightText: © 2022 ekvip automation GmbH <info@ekvip.de>
| SPDX-License-Identifier: Apache-2.0
| For details check: Apache-2.0_

.. _Apache-2.0: https://www.apache.org/licenses/LICENSE-2.0

.. </legal notes>

parameters
==========

*)

METHOD testAndMaskIsEqualTo 
VAR_INPUT
	(* for the test it's the parameter ``currentValue`` *)
	valueToTest	:LWORD;
	(* it's the mask for the currentValue *)
	mask		:LWORD;
	(* for the test it's the parameter ``expectedValue`` *)
	expected	:LWORD;
END_VAR
VAR
	(* just the expectation if the assertion to test must be worng or true *)
	assertionIsWrong		:BOOL;
	(* result of the bit operation to determine the value of ``assertionIsWrong`` *)
	result					:LWORD;
	(* contains the format string for the test message *)
	message					:Tc2_System.T_MaxString;
	(* TwinCAT printf with the test message *)
	messageStringBuilder	:Tc2_Utilities.FB_FormatString;
END_VAR
THIS^.assertorContainer.resetAssertor();

result := (valueToTest AND mask);
assertionIsWrong := (result <> expected);
message := SEL(
	assertionIsWrong,
	'currentValue: 16#%.16X AND mask: 16#%.16X is 16#%.16X expectedValue: 16#%.16X assertion must be TRUE', 
	'currentValue: 16#%.16X AND mask: 16#%.16X is 16#%.16X expectedValue: 16#%.16X assertion must be FALSE'
);
messageStringBuilder(
	sFormat := message,
	arg1 := THIS^.AnyToArg(valueToTest),
	arg2 := THIS^.AnyToArg(mask),
	arg3 := THIS^.AnyToArg(result),
	arg4 := THIS^.AnyToArg(expected)
);

THIS^.assertorContainer.assertor.assert.bitNumber.long.andMaskIsEqualTo(
	currentValue	:= valueToTest,
	mask 			:= mask,
	expectedValue	:= expected,
	message			:= ''
);

THIS^.AssertEquals_BOOL(
	Expected 	:= assertionIsWrong,
	Actual 		:= THIS^.assertorContainer.wasAssertionWrong,
	Message 	:= messageStringBuilder.sOut
);
END_METHOD

(*

long summary
==================
This test method tests ``assert.bitNumber.long.andMaskIsNotEqualTo``
method of CNM_AssertionInterfaces library, 
it provides the possibility to handover test data via parameter 


.. <legal notes>

legal notes
=================
| SPDX-FileCopyrightText: © 2022 ekvip automation GmbH <info@ekvip.de>
| SPDX-License-Identifier: Apache-2.0
| For details check: Apache-2.0_

.. _Apache-2.0: https://www.apache.org/licenses/LICENSE-2.0

.. </legal notes>

parameters
==========

*)

METHOD testAndMaskIsNotEqualTo 
VAR_INPUT
	(* for the test it's the parameter ``currentValue`` *)
	valueToTest	:LWORD;
	(* it's the mask for the currentValue *)
	mask		:LWORD;
	(* for the test it's the parameter ``unexpectedValue`` *)
	unexpected	:LWORD;
END_VAR
VAR
	(* just the expectation if the assertion to test must be worng or true *)
	assertionIsWrong		:BOOL;
	(* result of the bit operation to determine the value of ``assertionIsWrong`` *)
	result					:LWORD;
	(* contains the format string for the test message *)
	message					:Tc2_System.T_MaxString;
	(* TwinCAT printf with the test message *)
	messageStringBuilder	:Tc2_Utilities.FB_FormatString;
END_VAR
THIS^.assertorContainer.resetAssertor();

result := (valueToTest AND mask);
assertionIsWrong := (result = unexpected);
message := SEL(
	assertionIsWrong,
	'currentValue: 16#%.16X AND mask: 16#%.16X is 16#%.16X unexpectedValue: 16#%.16X assertion must be TRUE', 
	'currentValue: 16#%.16X AND mask: 16#%.16X is 16#%.16X unexpectedValue: 16#%.16X assertion must be FLASE'
);
messageStringBuilder(
	sFormat := message,
	arg1 := THIS^.AnyToArg(valueToTest),
	arg2 := THIS^.AnyToArg(mask),
	arg3 := THIS^.AnyToArg(result),
	arg4 := THIS^.AnyToArg(unexpected)
);

THIS^.assertorContainer.assertor.assert.bitNumber.long.andMaskIsNotEqualTo(
	currentValue	:= valueToTest,
	mask 			:= mask,
	unexpectedValue	:= unexpected,
	message			:= ''
);

THIS^.AssertEquals_BOOL(
	Expected 	:= assertionIsWrong,
	Actual 		:= THIS^.assertorContainer.wasAssertionWrong,
	Message 	:= messageStringBuilder.sOut
);
END_METHOD

(*

long summary
==================
This test method tests ``assert.bitNumber.long.bitXIsEqualTo``
method of CNM_AssertionInterfaces library, 
it provides the possibility to handover test data via parameter 


.. <legal notes>

legal notes
=================
| SPDX-FileCopyrightText: © 2022 ekvip automation GmbH <info@ekvip.de>
| SPDX-License-Identifier: Apache-2.0
| For details check: Apache-2.0_

.. _Apache-2.0: https://www.apache.org/licenses/LICENSE-2.0

.. </legal notes>

parameters
==========

*)

METHOD testBitXIsEqualTo
VAR_INPUT
	(* for the test it's the parameter ``currentValue`` *)
	valueToTest			:LWORD;
	(* the bit number to check in this test, it's the parameter ``number``*)
	bitNumberToCheck	:CNM_AssertionInterfaces.BitNumberLWord;
	(* this is the expected value of the bit ``bitNumberToCheck``, it's the parameter ``expectedValue`` *)
	bitIsSet			:BOOL;
END_VAR
VAR
	(* just the expectation if the assertion to test must be worng or true *)
	assertionIsWrong		:BOOL;
	(* bit with the number of ``bitNumberToCheck`` filtered from ``valueToTest`` *)
	specificBitOnly			:LWORD;
	(* the bit number ``bitNumberToCheck`` is set to the value of ``bitIsSet`` only *)
	testBitOnly				:LWORD;
	(* contains the format string for the test message *)
	message					:Tc2_System.T_MaxString;
	(* TwinCAT printf with the test message *)
	messageStringBuilder	:Tc2_Utilities.FB_FormatString;
END_VAR
THIS^.assertorContainer.resetAssertor();

specificBitOnly := (valueToTest AND SHL(THIS^.LSB_ONLY,bitNumberToCheck));
testBitOnly		:= SHL(TO_LWORD(bitIsSet),bitNumberToCheck);
assertionIsWrong := (specificBitOnly <> testBitOnly);

message := 'Bit number %d in currentValue: 16#%.16X ';
message := SEL(
	(specificBitOnly > THIS^.NO_BIT_SET),
	Tc2_Standard.CONCAT(message, 'is unset '),
	Tc2_Standard.CONCAT(message, 'is set ')
);
message := SEL(
	(testBitOnly > THIS^.NO_BIT_SET),
	Tc2_Standard.CONCAT(message, 'expectedValue: is unset (FALSE) '),
	Tc2_Standard.CONCAT(message, 'expectedValue: is set (TRUE)  ')
);
message := SEL(
	assertionIsWrong,
	Tc2_Standard.CONCAT(message, 'assertion must be TRUE'),
	Tc2_Standard.CONCAT(message, 'assertion must be FALSE')
);
messageStringBuilder(
	sFormat := message,
	arg1 := THIS^.AnyToArg(bitNumberToCheck),
	arg2 := THIS^.AnyToArg(valueToTest)
);


THIS^.assertorContainer.assertor.assert.bitNumber.long.bitXIsEqualTo(
	currentValue 	:= valueToTest,
	number			:= bitNumberToCheck,
	expectedValue	:= bitIsSet,
	message			:= ''  
); 

THIS^.AssertEquals_BOOL(
	Expected 	:= assertionIsWrong,
	Actual 		:= THIS^.assertorContainer.wasAssertionWrong,
	Message 	:= messageStringBuilder.sOut
);
END_METHOD

(*

long summary
==================
This test method tests ``assert.bitNumber.long.bitXIsNotEqualTo``
method of CNM_AssertionInterfaces library, 
it provides the possibility to handover test data via parameter 


.. <legal notes>

legal notes
=================
| SPDX-FileCopyrightText: © 2022 ekvip automation GmbH <info@ekvip.de>
| SPDX-License-Identifier: Apache-2.0
| For details check: Apache-2.0_

.. _Apache-2.0: https://www.apache.org/licenses/LICENSE-2.0

.. </legal notes>

parameters
==========

*)

METHOD testBitXIsNotEqualTo
VAR_INPUT
	(* for the test it's the parameter ``currentValue`` *)
	valueToTest			:LWORD;
	(* the bit number to check in this test, it's the parameter ``number``*)
	bitNumberToCheck	:CNM_AssertionInterfaces.BitNumberLWord;
	(* this is the unexpected value of the bit ``bitNumberToCheck``, it's the parameter ``unexpectedValue`` *)
	bitIsSet			:BOOL;
END_VAR
VAR
	(* just the expectation if the assertion to test must be worng or true *)
	assertionIsWrong		:BOOL;
	(* bit with the number of ``bitNumberToCheck`` filtered from ``valueToTest`` *)
	specificBitOnly			:LWORD;
	(* the bit number ``bitNumberToCheck`` is set to the value of ``bitIsSet`` only *)
	testBitOnly				:LWORD;
	(* contains the format string for the test message *)
	message					:Tc2_System.T_MaxString;
	(* TwinCAT printf with the test message *)
	messageStringBuilder	:Tc2_Utilities.FB_FormatString;
END_VAR
THIS^.assertorContainer.resetAssertor();

specificBitOnly := (valueToTest AND SHL(THIS^.LSB_ONLY,bitNumberToCheck));
testBitOnly		:= SHL(TO_LWORD(bitIsSet),bitNumberToCheck);
assertionIsWrong := (specificBitOnly = testBitOnly);

message := 'Bit number %d in currentValue: 16#%.16X ';
message := SEL(
	(specificBitOnly > THIS^.NO_BIT_SET),
	Tc2_Standard.CONCAT(message, 'is unset '),
	Tc2_Standard.CONCAT(message, 'is set ')
);
message := SEL(
	(testBitOnly > THIS^.NO_BIT_SET),
	Tc2_Standard.CONCAT(message, 'unexpectedValue: is unset (FALSE) '),
	Tc2_Standard.CONCAT(message, 'unexpectedValue: is set (TRUE)  ')
);
message := SEL(
	assertionIsWrong,
	Tc2_Standard.CONCAT(message, 'assertion must be TRUE'),
	Tc2_Standard.CONCAT(message, 'assertion must be FALSE')
);
messageStringBuilder(
	sFormat := message,
	arg1 := THIS^.AnyToArg(bitNumberToCheck),
	arg2 := THIS^.AnyToArg(valueToTest)
);

THIS^.assertorContainer.assertor.assert.bitNumber.long.bitXIsNotEqualTo(
	currentValue 	:= valueToTest,
	number			:= bitNumberToCheck,
	unexpectedValue	:= bitIsSet,
	message			:= ''  
); 

THIS^.AssertEquals_BOOL(
	Expected 	:= assertionIsWrong,
	Actual 		:= THIS^.assertorContainer.wasAssertionWrong,
	Message 	:= messageStringBuilder.sOut
);
END_METHOD

(*

long summary
==================
This test method tests ``assert.bitNumber.long.bitXIsSet``
of CNM_AssertionInterfaces library, 
it provides the possibility to handover test data via parameter 


.. <legal notes>

legal notes
=================
| SPDX-FileCopyrightText: © 2022 ekvip automation GmbH <info@ekvip.de>
| SPDX-License-Identifier: Apache-2.0
| For details check: Apache-2.0_

.. _Apache-2.0: https://www.apache.org/licenses/LICENSE-2.0

.. </legal notes>

parameters
==========

*)

METHOD testBitXIsSet
VAR_INPUT
	(* for the test it's the parameter ``currentValue`` *)
	valueToTest			:LWORD;
	(* the bit number to check in this test, it's the parameter ``number``*)
	bitNumberToCheck	:CNM_AssertionInterfaces.BitNumberLWord;
END_VAR
VAR
	(* just the expectation if the assertion to test must be worng or true *)
	assertionIsWrong		:BOOL;
	(* contains the format string for the test message *)
	message					:Tc2_System.T_MaxString;
	(* TwinCAT printf with the test message *)
	messageStringBuilder	:Tc2_Utilities.FB_FormatString;
END_VAR
THIS^.assertorContainer.resetAssertor();

assertionIsWrong := ((valueToTest AND SHL(THIS^.LSB_ONLY,bitNumberToCheck)) = THIS^.NO_BIT_SET);

message := SEL(
	assertionIsWrong,
	'Bit number %d in currentValue: 16#%.16X is set assertion must be TRUE',
	'Bit number %d in currentValue: 16#%.16X is unset assertion must be FALSE'
);

messageStringBuilder(
	sFormat := message,
	arg1 := THIS^.AnyToArg(bitNumberToCheck),
	arg2 := THIS^.AnyToArg(valueToTest)
);

THIS^.assertorContainer.assertor.assert.bitNumber.long.bitXIsSet(
	currentValue := valueToTest,
	number := bitNumberToCheck,
	message := ''
);

THIS^.AssertEquals_BOOL(
	Expected 	:= assertionIsWrong,
	Actual 		:= THIS^.assertorContainer.wasAssertionWrong,
	Message 	:= messageStringBuilder.sOut
);
END_METHOD

(*

long summary
==================
This test method tests ``assert.bitNumber.long.bitXIsUnset``
of CNM_AssertionInterfaces library, 
it provides the possibility to handover test data via parameter 


.. <legal notes>

legal notes
=================
| SPDX-FileCopyrightText: © 2022 ekvip automation GmbH <info@ekvip.de>
| SPDX-License-Identifier: Apache-2.0
| For details check: Apache-2.0_

.. _Apache-2.0: https://www.apache.org/licenses/LICENSE-2.0

.. </legal notes>

parameters
==========

*)

METHOD testBitXIsUnset
VAR_INPUT
	(* for the test it's the parameter ``currentValue`` *)
	valueToTest			:LWORD;
	(* the bit number to check in this test, it's the parameter ``number``*)
	bitNumberToCheck	:CNM_AssertionInterfaces.BitNumberLWord;
END_VAR
VAR
	(* just the expectation if the assertion to test must be worng or true *)
	assertionIsWrong		:BOOL;
	(* contains the format string for the test message *)
	message					:Tc2_System.T_MaxString;
	(* TwinCAT printf with the test message *)
	messageStringBuilder	:Tc2_Utilities.FB_FormatString;
END_VAR
THIS^.assertorContainer.resetAssertor();

assertionIsWrong := ((valueToTest AND SHL(THIS^.LSB_ONLY,bitNumberToCheck)) > THIS^.NO_BIT_SET);

message := SEL(
	assertionIsWrong,
	'Bit number %d in currentValue: 16#%.16X is unset assertion must be TRUE',
	'Bit number %d in currentValue: 16#%.16X is set assertion must be FALSE'
);

messageStringBuilder(
	sFormat := message,
	arg1 := THIS^.AnyToArg(bitNumberToCheck),
	arg2 := THIS^.AnyToArg(valueToTest)
);

THIS^.assertorContainer.assertor.assert.bitNumber.long.bitXIsUnset(
	currentValue := valueToTest,
	number := bitNumberToCheck,
	message := ''
);

THIS^.AssertEquals_BOOL(
	Expected 	:= assertionIsWrong,
	Actual 		:= THIS^.assertorContainer.wasAssertionWrong,
	Message 	:= messageStringBuilder.sOut
);
END_METHOD

(*

long summary
==================
This test method tests ``assert.bitNumber.long.lsbIsEqualTo``
method of CNM_AssertionInterfaces library, 
it provides the possibility to handover test data via parameter 


.. <legal notes>

legal notes
=================
| SPDX-FileCopyrightText: © 2022 ekvip automation GmbH <info@ekvip.de>
| SPDX-License-Identifier: Apache-2.0
| For details check: Apache-2.0_

.. _Apache-2.0: https://www.apache.org/licenses/LICENSE-2.0

.. </legal notes>

parameters
==========

*)

METHOD testLsbIsEqualTo
VAR_INPUT
	(* for the test it's the parameter ``currentValue`` *)
	valueToTest		:LWORD;
	(* for the test it's the parameter ``expectedValue`` *)
	expectedValue	:BOOL;
END_VAR
VAR
	(* just the expectation if the assertion to test must be worng or true *)
	assertionIsWrong		:BOOL;
	(* contains the format string for the test message *)
	message					:Tc2_System.T_MaxString;
	(* TwinCAT printf with the test message *)
	messageStringBuilder	:Tc2_Utilities.FB_FormatString;
END_VAR
THIS^.assertorContainer.resetAssertor();

assertionIsWrong := (valueToTest.FIRST_BIT <> expectedValue);
message := SEL(
	expectedValue,
	'currentValue: %d expectedValue is an unset (FALSE) assertion must be ',
	'currentValue: %d expectedValue is a set (TRUE) assertion must be '
);
message := SEL(
	assertionIsWrong,
	Tc2_Standard.CONCAT(message, 'TRUE'),
	Tc2_Standard.CONCAT(message, 'FALSE')
);

messageStringBuilder(
	sFormat := message,
	arg1 := THIS^.AnyToArg(valueToTest)
);

THIS^.assertorContainer.assertor.assert.bitNumber.long.lsbIsEqualTo(
	currentValue 	:= valueToTest,
	expectedValue	:= expectedValue,
	message			:= ''  
); 

THIS^.AssertEquals_BOOL(
	Expected 	:= assertionIsWrong,
	Actual 		:= THIS^.assertorContainer.wasAssertionWrong,
	Message 	:= messageStringBuilder.sOut
);
END_METHOD

(*

long summary
==================
This test method tests ``assert.bitNumber.long.lsbIsNotEqualTo``
method of CNM_AssertionInterfaces library, 
it provides the possibility to handover test data via parameter 


.. <legal notes>

legal notes
=================
| SPDX-FileCopyrightText: © 2022 ekvip automation GmbH <info@ekvip.de>
| SPDX-License-Identifier: Apache-2.0
| For details check: Apache-2.0_

.. _Apache-2.0: https://www.apache.org/licenses/LICENSE-2.0

.. </legal notes>

parameters
==========

*)

METHOD testLsbIsNotEqualTo
VAR_INPUT
	(* for the test it's the parameter ``currentValue`` *)
	valueToTest	:LWORD;
	(* for the test it's the parameter ``unexpectedValue`` *)
	unexpectedValue :BOOL;
END_VAR
VAR
	(* just the expectation if the assertion to test must be worng or true *)
	assertionIsWrong		:BOOL;
	(* contains the format string for the test message *)
	message					:Tc2_System.T_MaxString;
	(* TwinCAT printf with the test message *)
	messageStringBuilder	:Tc2_Utilities.FB_FormatString;
END_VAR
THIS^.assertorContainer.resetAssertor();

assertionIsWrong := (valueToTest.FIRST_BIT = unexpectedValue);
message := SEL(
	unexpectedValue,
	'currentValue: %d unexpectedValue is an unset (FALSE), assertion must be ',
	'currentValue: %d unexpectedValue is a set (TRUE) assertion must be '
);
message := SEL(
	assertionIsWrong,
	Tc2_Standard.CONCAT(message, 'TRUE'),
	Tc2_Standard.CONCAT(message, 'FALSE')
);

messageStringBuilder(
	sFormat := message,
	arg1 := THIS^.AnyToArg(valueToTest)
);

THIS^.assertorContainer.assertor.assert.bitNumber.long.lsbIsNotEqualTo(
	currentValue 	:= valueToTest,
	unexpectedValue	:= unexpectedValue,
	message			:= ''  
); 

THIS^.AssertEquals_BOOL(
	Expected 	:= assertionIsWrong,
	Actual 		:= THIS^.assertorContainer.wasAssertionWrong,
	Message 	:= messageStringBuilder.sOut
);
END_METHOD

(*

long summary
==================
This test method tests ``assert.bitNumber.long.lsbIsSet``
of CNM_AssertionInterfaces library, 
it provides the possibility to handover test data via parameter 


.. <legal notes>

legal notes
=================
| SPDX-FileCopyrightText: © 2022 ekvip automation GmbH <info@ekvip.de>
| SPDX-License-Identifier: Apache-2.0
| For details check: Apache-2.0_

.. _Apache-2.0: https://www.apache.org/licenses/LICENSE-2.0

.. </legal notes>

parameters
==========

*)

METHOD testLsbIsSet
VAR_INPUT
	(* for the test it's the parameter ``currentValue`` *)
	valueToTest	:LWORD;
END_VAR
VAR
	(* just the expectation if the assertion to test must be worng or true *)
	assertionIsWrong		:BOOL;
	(* contains the format string for the test message *)
	message					:Tc2_System.T_MaxString;
	(* TwinCAT printf with the test message *)
	messageStringBuilder	:Tc2_Utilities.FB_FormatString;
END_VAR
THIS^.assertorContainer.resetAssertor();

assertionIsWrong := (NOT valueToTest.FIRST_BIT);

message := SEL(
	assertionIsWrong,
	'currentValue is %d assertion must be TRUE',
	'currentValue is %d assertion must be FALSE'
);

messageStringBuilder(
	sFormat := message,
	arg1 := THIS^.AnyToArg(valueToTest)
);

THIS^.assertorContainer.assertor.assert.bitNumber.long.lsbIsSet(
	currentValue 	:= valueToTest,
	message			:= ''  
); 

THIS^.AssertEquals_BOOL(
	Expected 	:= assertionIsWrong,
	Actual 		:= THIS^.assertorContainer.wasAssertionWrong,
	Message 	:= messageStringBuilder.sOut
);
END_METHOD

(*

long summary
==================
This test method tests ``assert.bitNumber.long.lsbIsUnset``
and ``assert.bitNumber.long.lsbIsUnset``
of CNM_AssertionInterfaces library, 
it provides the possibility to handover test data via parameter 


.. <legal notes>

legal notes
=================
| SPDX-FileCopyrightText: © 2022 ekvip automation GmbH <info@ekvip.de>
| SPDX-License-Identifier: Apache-2.0
| For details check: Apache-2.0_

.. _Apache-2.0: https://www.apache.org/licenses/LICENSE-2.0

.. </legal notes>

parameters
==========

*)

METHOD testLsbIsUnset
VAR_INPUT
	(* for the test it's the parameter ``currentValue`` *)
	valueToTest	:LWORD;
END_VAR
VAR
	(* just the expectation if the assertion to test must be worng or true *)
	assertionIsWrong		:BOOL;
	(* contains the format string for the test message *)
	message					:Tc2_System.T_MaxString;
	(* TwinCAT printf with the test message *)
	messageStringBuilder	:Tc2_Utilities.FB_FormatString;
END_VAR
THIS^.assertorContainer.resetAssertor();

assertionIsWrong := (valueToTest.FIRST_BIT);

message := SEL(
	assertionIsWrong,
	'currentValue is %d assertion must be TRUE',
	'currentValue is %d assertion must be FALSE'
);

messageStringBuilder(
	sFormat := message,
	arg1 := THIS^.AnyToArg(valueToTest)
);

THIS^.assertorContainer.assertor.assert.bitNumber.long.lsbIsUnset(
	currentValue 	:= valueToTest,
	message			:= ''  
); 

THIS^.AssertEquals_BOOL(
	Expected 	:= assertionIsWrong,
	Actual 		:= THIS^.assertorContainer.wasAssertionWrong,
	Message 	:= messageStringBuilder.sOut
);
END_METHOD

(*

long summary
==================
This test method tests ``assert.bitNumber.long.msbIsEqualTo``
method of CNM_AssertionInterfaces library, 
it provides the possibility to handover test data via parameter 


.. <legal notes>

legal notes
=================
| SPDX-FileCopyrightText: © 2022 ekvip automation GmbH <info@ekvip.de>
| SPDX-License-Identifier: Apache-2.0
| For details check: Apache-2.0_

.. _Apache-2.0: https://www.apache.org/licenses/LICENSE-2.0

.. </legal notes>

parameters
==========

*)

METHOD testMsbIsEqualTo
VAR_INPUT
	(* for the test it's the parameter ``currentValue`` *)
	valueToTest		:LWORD;
	(* for the test it's the parameter ``expectedValue`` *)
	expectedValue	:BOOL;
END_VAR
VAR
	(* just the expectation if the assertion to test must be worng or true *)
	assertionIsWrong		:BOOL;
	(* contains the format string for the test message *)
	message					:Tc2_System.T_MaxString;
	(* TwinCAT printf with the test message *)
	messageStringBuilder	:Tc2_Utilities.FB_FormatString;
END_VAR
THIS^.assertorContainer.resetAssertor();

assertionIsWrong := (valueToTest.LAST_BIT <> expectedValue);

message := SEL(
	expectedValue,
	'currentValue: 16#%.16X expectedValue is an unset (FALSE) assertion must be ',
	'currentValue: 16#%.16X expectedValue is a set (TRUE) assertion must be '
);
message := SEL(
	assertionIsWrong,
	Tc2_Standard.CONCAT(message, 'TRUE'),
	Tc2_Standard.CONCAT(message, 'FALSE')
);

messageStringBuilder(
	sFormat := message,
	arg1 := THIS^.AnyToArg(valueToTest)
);

THIS^.assertorContainer.assertor.assert.bitNumber.long.msbIsEqualTo(
	currentValue 	:= valueToTest,
	expectedValue	:= expectedValue,
	message			:= ''  
); 

THIS^.AssertEquals_BOOL(
	Expected 	:= assertionIsWrong,
	Actual 		:= THIS^.assertorContainer.wasAssertionWrong,
	Message 	:= messageStringBuilder.sOut
);
END_METHOD

(*

long summary
==================
This test method tests ``assert.bitNumber.long.msbIsNotEqualTo``
method of CNM_AssertionInterfaces library, 
it provides the possibility to handover test data via parameter 


.. <legal notes>

legal notes
=================
| SPDX-FileCopyrightText: © 2022 ekvip automation GmbH <info@ekvip.de>
| SPDX-License-Identifier: Apache-2.0
| For details check: Apache-2.0_

.. _Apache-2.0: https://www.apache.org/licenses/LICENSE-2.0

.. </legal notes>

parameters
==========

*)

METHOD testMsbIsNotEqualTo
VAR_INPUT
	(* for the test it's the parameter ``currentValue`` *)
	valueToTest	:LWORD;
	(* for the test it's the parameter ``unexpectedValue`` *)
	unexpectedValue :BOOL;
END_VAR
VAR
	(* just the expectation if the assertion to test must be worng or true *)
	assertionIsWrong		:BOOL;
	(* contains the format string for the test message *)
	message					:Tc2_System.T_MaxString;
	(* TwinCAT printf with the test message *)
	messageStringBuilder	:Tc2_Utilities.FB_FormatString;
END_VAR
THIS^.assertorContainer.resetAssertor();

assertionIsWrong := (valueToTest.LAST_BIT = unexpectedValue);

message := SEL(
	unexpectedValue,
	'currentValue: 16#%.16X unexpectedValue is an unset (FALSE) assertion must be ',
	'currentValue: 16#%.16X unexpectedValue is a set (TRUE) assertion must be '
);
message := SEL(
	assertionIsWrong,
	Tc2_Standard.CONCAT(message, 'TRUE'),
	Tc2_Standard.CONCAT(message, 'FALSE')
);

messageStringBuilder(
	sFormat := message,
	arg1 := THIS^.AnyToArg(valueToTest)
);

THIS^.assertorContainer.assertor.assert.bitNumber.long.msbIsNotEqualTo(
	currentValue 	:= valueToTest,
	unexpectedValue	:= unexpectedValue,
	message			:= ''  
); 

THIS^.AssertEquals_BOOL(
	Expected 	:= assertionIsWrong,
	Actual 		:= THIS^.assertorContainer.wasAssertionWrong,
	Message 	:= messageStringBuilder.sOut
);
END_METHOD

(*

long summary
==================
This test method tests ``assert.bitNumber.long.msbIsSet``
of CNM_AssertionInterfaces library, 
it provides the possibility to handover test data via parameter 


.. <legal notes>

legal notes
=================
| SPDX-FileCopyrightText: © 2022 ekvip automation GmbH <info@ekvip.de>
| SPDX-License-Identifier: Apache-2.0
| For details check: Apache-2.0_

.. _Apache-2.0: https://www.apache.org/licenses/LICENSE-2.0

.. </legal notes>

parameters
==========

*)

METHOD testMsbIsSet
VAR_INPUT
	(* for the test it's the parameter ``currentValue`` *)
	valueToTest	:LWORD;
END_VAR
VAR
	(* just the expectation if the assertion to test must be worng or true *)
	assertionIsWrong		:BOOL;
	(* contains the format string for the test message *)
	message					:Tc2_System.T_MaxString;
	(* TwinCAT printf with the test message *)
	messageStringBuilder	:Tc2_Utilities.FB_FormatString;
END_VAR
THIS^.assertorContainer.resetAssertor();

assertionIsWrong := (NOT valueToTest.LAST_BIT);

message := SEL(
	assertionIsWrong,
	'currentValue is 16#%.16X assertion must be TRUE',
	'currentValue is 16#%.16X assertion must be FALSE'
);

messageStringBuilder(
	sFormat := message,
	arg1 := THIS^.AnyToArg(valueToTest)
);

THIS^.assertorContainer.assertor.assert.bitNumber.long.msbIsSet(
	currentValue 	:= valueToTest,
	message			:= ''  
); 

THIS^.AssertEquals_BOOL(
	Expected 	:= assertionIsWrong,
	Actual 		:= THIS^.assertorContainer.wasAssertionWrong,
	Message 	:= messageStringBuilder.sOut
);
END_METHOD

(*

long summary
==================
This test method tests ``assert.bitNumber.long.msbIsUnset``
of CNM_AssertionInterfaces library, 
it provides the possibility to handover test data via parameter 


.. <legal notes>

legal notes
=================
| SPDX-FileCopyrightText: © 2022 ekvip automation GmbH <info@ekvip.de>
| SPDX-License-Identifier: Apache-2.0
| For details check: Apache-2.0_

.. _Apache-2.0: https://www.apache.org/licenses/LICENSE-2.0

.. </legal notes>

parameters
==========

*)

METHOD testMsbIsUnset
VAR_INPUT
	(* for the test it's the parameter ``currentValue`` *)
	valueToTest	:LWORD;
END_VAR
VAR
	(* just the expectation if the assertion to test must be worng or true *)
	assertionIsWrong		:BOOL;
	(* contains the format string for the test message *)
	message					:Tc2_System.T_MaxString;
	(* TwinCAT printf with the test message *)
	messageStringBuilder	:Tc2_Utilities.FB_FormatString;
END_VAR
THIS^.assertorContainer.resetAssertor();

assertionIsWrong := (valueToTest.LAST_BIT);

message := SEL(
	assertionIsWrong,
	'currentValue is 16#%.16X assertion must be TRUE',
	'currentValue is 16#%.16X assertion must be FALSE'
);

messageStringBuilder(
	sFormat := message,
	arg1 := THIS^.AnyToArg(valueToTest)
);

THIS^.assertorContainer.assertor.assert.bitNumber.long.msbIsUnset(
	currentValue 	:= valueToTest,
	message			:= ''  
); 

THIS^.AssertEquals_BOOL(
	Expected 	:= assertionIsWrong,
	Actual 		:= THIS^.assertorContainer.wasAssertionWrong,
	Message 	:= messageStringBuilder.sOut
);
END_METHOD

(*

long summary
==================
This test method tests ``assert.bitNumber.long.orMaskIsEqualTo``
method of CNM_AssertionInterfaces library, 
it provides the possibility to handover test data via parameter 


.. <legal notes>

legal notes
=================
| SPDX-FileCopyrightText: © 2022 ekvip automation GmbH <info@ekvip.de>
| SPDX-License-Identifier: Apache-2.0
| For details check: Apache-2.0_

.. _Apache-2.0: https://www.apache.org/licenses/LICENSE-2.0

.. </legal notes>

parameters
==========

*)

METHOD testOrMaskIsEqualTo 
VAR_INPUT
	(* for the test it's the parameter ``currentValue`` *)
	valueToTest	:LWORD;
	(* it's the mask for the currentValue *)
	mask		:LWORD;
	(* for the test it's the parameter ``expectedValue`` *)
	expected	:LWORD;
END_VAR
VAR
	(* just the expectation if the assertion to test must be worng or true *)
	assertionIsWrong		:BOOL;
	(* result of the bit operation to determine the value of ``assertionIsWrong`` *)
	result					:LWORD;
	(* contains the format string for the test message *)
	message					:Tc2_System.T_MaxString;
	(* TwinCAT printf with the test message *)
	messageStringBuilder	:Tc2_Utilities.FB_FormatString;
END_VAR
THIS^.assertorContainer.resetAssertor();

result := (valueToTest OR mask);
assertionIsWrong := (result <> expected);
message := SEL(
	assertionIsWrong,
	'currentValue: 16#%.16X OR mask: 16#%.16X is 16#%.16X expectedValue: 16#%.16X assertion must be TRUE', 
	'currentValue: 16#%.16X OR mask: 16#%.16X is 16#%.16X expectedValue: 16#%.16X assertion must be FALSE'
);
messageStringBuilder(
	sFormat := message,
	arg1 := THIS^.AnyToArg(valueToTest),
	arg2 := THIS^.AnyToArg(mask),
	arg3 := THIS^.AnyToArg(result),
	arg4 := THIS^.AnyToArg(expected)
);

THIS^.assertorContainer.assertor.assert.bitNumber.long.orMaskIsEqualTo(
	currentValue	:= valueToTest,
	mask 			:= mask,
	expectedValue	:= expected,
	message			:= ''
);

THIS^.AssertEquals_BOOL(
	Expected 	:= assertionIsWrong,
	Actual 		:= THIS^.assertorContainer.wasAssertionWrong,
	Message 	:= messageStringBuilder.sOut
);
END_METHOD

(*

long summary
==================
This test method tests ``assert.bitNumber.long.orMaskIsNotEqualTo``
method of CNM_AssertionInterfaces library, 
it provides the possibility to handover test data via parameter 


.. <legal notes>

legal notes
=================
| SPDX-FileCopyrightText: © 2022 ekvip automation GmbH <info@ekvip.de>
| SPDX-License-Identifier: Apache-2.0
| For details check: Apache-2.0_

.. _Apache-2.0: https://www.apache.org/licenses/LICENSE-2.0

.. </legal notes>

parameters
==========

*)

METHOD testOrMaskIsNotEqualTo 
VAR_INPUT
	(* for the test it's the parameter ``currentValue`` *)
	valueToTest	:LWORD;
	(* it's the mask for the currentValue *)
	mask		:LWORD;
	(* for the test it's the parameter ``unexpectedValue`` *)
	unexpected	:LWORD;
END_VAR
VAR
	(* just the expectation if the assertion to test must be worng or true *)
	assertionIsWrong		:BOOL;
	(* result of the bit operation to determine the value of ``assertionIsWrong`` *)
	result					:LWORD;
	(* contains the format string for the test message *)
	message					:Tc2_System.T_MaxString;
	(* TwinCAT printf with the test message *)
	messageStringBuilder	:Tc2_Utilities.FB_FormatString;
END_VAR
THIS^.assertorContainer.resetAssertor();

result := (valueToTest OR mask);
assertionIsWrong := (result = unexpected);
message := SEL(
	assertionIsWrong,
	'currentValue: 16#%.16X OR mask: 16#%.16X is 16#%.16X unexpectedValue: 16#%.16X assertion must be TRUE', 
	'currentValue: 16#%.16X OR mask: 16#%.16X is 16#%.16X unexpectedValue: 16#%.16X assertion must be FALSE'
);
messageStringBuilder(
	sFormat := message,
	arg1 := THIS^.AnyToArg(valueToTest),
	arg2 := THIS^.AnyToArg(mask),
	arg3 := THIS^.AnyToArg(result),
	arg4 := THIS^.AnyToArg(unexpected)
);

THIS^.assertorContainer.assertor.assert.bitNumber.long.orMaskIsNotEqualTo(
	currentValue	:= valueToTest,
	mask 			:= mask,
	unexpectedValue	:= unexpected,
	message			:= ''
);

THIS^.AssertEquals_BOOL(
	Expected 	:= assertionIsWrong,
	Actual 		:= THIS^.assertorContainer.wasAssertionWrong,
	Message 	:= messageStringBuilder.sOut
);
END_METHOD

(*

long summary
==================
This test method tests ``assert.bitNumber.long.valueIsEqualTo``
method of CNM_AssertionInterfaces library, 
it provides the possibility to handover test data via parameter 


.. <legal notes>

legal notes
=================
| SPDX-FileCopyrightText: © 2022 ekvip automation GmbH <info@ekvip.de>
| SPDX-License-Identifier: Apache-2.0
| For details check: Apache-2.0_

.. _Apache-2.0: https://www.apache.org/licenses/LICENSE-2.0

.. </legal notes>

parameters
==========

*)

METHOD testValueIsEqualTo
VAR_INPUT
	(* for the test it's the parameter ``currentValue`` *)
	valueToTest	:LWORD;
	(* for the test it's the parameter ``expectedValue`` *)
	expected	:LWORD;
END_VAR
VAR
	(* just the expectation if the assertion to test must be worng or true *)
	assertionIsWrong		:BOOL;
	(* contains the format string for the test message *)
	message					:Tc2_System.T_MaxString;
	(* TwinCAT printf with the test message *)
	messageStringBuilder	:Tc2_Utilities.FB_FormatString;
END_VAR
THIS^.assertorContainer.resetAssertor();

assertionIsWrong := (valueToTest <> expected);
message := SEL(
	assertionIsWrong,
	'currentValue is %d expectedValue is %d assertion must be TRUE', 
	'currentValue is %d expectedValue is %d assertion must be FALSE'
);
messageStringBuilder(
	sFormat := message,
	arg1 := THIS^.AnyToArg(valueToTest),
	arg2 := THIS^.AnyToArg(expected)
);

THIS^.assertorContainer.assertor.assert.bitNumber.long.valueIsEqualTo(
	currentValue := valueToTest,
	expectedValue := expected,
	message := ''
);

THIS^.AssertEquals_BOOL(
	Expected 	:= assertionIsWrong,
	Actual 		:= THIS^.assertorContainer.wasAssertionWrong,
	Message 	:= messageStringBuilder.sOut
);
END_METHOD

(*

long summary
==================
This test method tests ``assert.bitNumber.long.valueIsGreaterThan``
method of CNM_AssertionInterfaces library, 
it provides the possibility to handover test data via parameter 


.. <legal notes>

legal notes
=================
| SPDX-FileCopyrightText: © 2022 ekvip automation GmbH <info@ekvip.de>
| SPDX-License-Identifier: Apache-2.0
| For details check: Apache-2.0_

.. _Apache-2.0: https://www.apache.org/licenses/LICENSE-2.0

.. </legal notes>

parameters
==========

*)

METHOD testValueIsGreater
VAR_INPUT
	(* for the test it's the parameter ``currentValue`` *)
	valueToTest	:LWORD;
	(* for the test it's the parameter ``lessValue`` *)
	less		:LWORD;
END_VAR
VAR
	(* just the expectation if the assertion to test must be worng or true *)
	assertionIsWrong		:BOOL;
	(* contains the format string for the test message *)
	message					:Tc2_System.T_MaxString;
	(* TwinCAT printf with the test message *)
	messageStringBuilder	:Tc2_Utilities.FB_FormatString;
END_VAR
THIS^.assertorContainer.resetAssertor();

assertionIsWrong := (valueToTest <= less);
message := SEL(
	assertionIsWrong,
	'currentValue is %d lessValue is %d assertion must be TRUE', 
	'currentValue is %d lessValue is %d assertion must be FALSE'
);
messageStringBuilder(
	sFormat := message,
	arg1 := THIS^.AnyToArg(valueToTest),
	arg2 := THIS^.AnyToArg(less)
);

THIS^.assertorContainer.assertor.assert.bitNumber.long.valueIsGreaterThan(
	currentValue := valueToTest,
	lessValue := less,
	message := ''
);

THIS^.AssertEquals_BOOL(
	Expected 	:= assertionIsWrong,
	Actual 		:= THIS^.assertorContainer.wasAssertionWrong,
	Message 	:= messageStringBuilder.sOut
);
END_METHOD

(*

long summary
==================
This test method tests ``assert.bitNumber.long.valueIsInRangeOf``
method of CNM_AssertionInterfaces library, 
it provides the possibility to handover test data via parameter 


.. <legal notes>

legal notes
=================
| SPDX-FileCopyrightText: © 2022 ekvip automation GmbH <info@ekvip.de>
| SPDX-License-Identifier: Apache-2.0
| For details check: Apache-2.0_

.. _Apache-2.0: https://www.apache.org/licenses/LICENSE-2.0

.. </legal notes>

parameters
==========

*)

METHOD testValueIsInRangeOf
VAR_INPUT
	(* for the test it's the parameter ``lowerLimit`` *)
	lower		:LWORD;
	(* for the test it's the parameter ``currentValue`` *)
	valueToTest	:LWORD;
	(* for the test it's the parameter ``upperLimit`` *)
	upper		:LWORD;
END_VAR          
VAR
	(* just the expectation if the assertion to test must be worng or true *)
	assertionIsWrong		:BOOL;
	(* contains the format string for the test message *)
	message					:Tc2_System.T_MaxString;
	(* TwinCAT printf with the test message *)
	messageStringBuilder	:Tc2_Utilities.FB_FormatString;
END_VAR
THIS^.assertorContainer.resetAssertor();

assertionIsWrong := ((valueToTest < lower) OR (valueToTest > upper)); 

message := SEL(
	assertionIsWrong,
	'lowerLimit is %d currentValue is %d upperLimit is %d assertion must be TRUE', 
	'lowerLimit is %d currentValue is %d upperLimit is %d assertion must be FALSE'
);

messageStringBuilder(
	sFormat := message,
	arg1 := THIS^.AnyToArg(lower),
	arg2 := THIS^.AnyToArg(valueToTest),
	arg3 := THIS^.AnyToArg(upper)
);

THIS^.assertorContainer.assertor.assert.bitNumber.long.valueIsInRangeOf(
	lowerLimit := lower,
	currentValue := valueToTest,
	upperLimit := upper,
	message := ''
);

THIS^.AssertEquals_BOOL(
	Expected 	:= assertionIsWrong,
	Actual 		:= THIS^.assertorContainer.wasAssertionWrong,
	Message 	:= messageStringBuilder.sOut
);
END_METHOD

(*

long summary
==================
This test method tests ``assert.bitNumber.long.valueIsLessThan``
method of CNM_AssertionInterfaces library, 
it provides the possibility to handover test data via parameter 


.. <legal notes>

legal notes
=================
| SPDX-FileCopyrightText: © 2022 ekvip automation GmbH <info@ekvip.de>
| SPDX-License-Identifier: Apache-2.0
| For details check: Apache-2.0_

.. _Apache-2.0: https://www.apache.org/licenses/LICENSE-2.0

.. </legal notes>

parameters
==========

*)

METHOD testValueIsLessThan
VAR_INPUT
	(* for the test it's the parameter ``currentValue`` *)
	valueToTest	:LWORD;
	(* for the test it's the parameter ``greaterValue`` *)
	greater		:LWORD;
END_VAR
VAR
	(* just the expectation if the assertion to test must be worng or true *)
	assertionIsWrong		:BOOL;
	(* contains the format string for the test message *)
	message					:Tc2_System.T_MaxString;
	(* TwinCAT printf with the test message *)
	messageStringBuilder	:Tc2_Utilities.FB_FormatString;
END_VAR
THIS^.assertorContainer.resetAssertor();

assertionIsWrong := (valueToTest >= greater);
message := SEL(
	assertionIsWrong,
	'currentValue is %d greaterValue is %d assertion must be TRUE',
	'currentValue is %d greaterValue is %d assertion must be FALSE'
);
messageStringBuilder(
	sFormat := message,
	arg1 := THIS^.AnyToArg(valueToTest),
	arg2 := THIS^.AnyToArg(greater)
);

THIS^.assertorContainer.assertor.assert.bitNumber.long.valueIsLessThan(
	currentValue := valueToTest,
	greaterValue := greater,
	message := ''
);

THIS^.AssertEquals_BOOL(
	Expected 	:= assertionIsWrong,
	Actual 		:= THIS^.assertorContainer.wasAssertionWrong,
	Message 	:= messageStringBuilder.sOut
);
END_METHOD

(*

long summary
==================
This test method tests ``assert.bitNumber.long.valueIsMax``
method of CNM_AssertionInterfaces library, 
it provides the possibility to handover test data via parameter 


.. <legal notes>

legal notes
=================
| SPDX-FileCopyrightText: © 2022 ekvip automation GmbH <info@ekvip.de>
| SPDX-License-Identifier: Apache-2.0
| For details check: Apache-2.0_

.. _Apache-2.0: https://www.apache.org/licenses/LICENSE-2.0

.. </legal notes>

parameters
==========

*)

METHOD testValueIsMax 
VAR_INPUT
	(* for the test it's the parameter ``currentValue`` *)
	valueToTest	:LWORD;
	(* for the test it's the parameter ``maximumValue`` *)
	maximum		:LWORD;
END_VAR
VAR
	(* just the expectation if the assertion to test must be worng or true *)
	assertionIsWrong		:BOOL;
	(* contains the format string for the test message *)
	message					:Tc2_System.T_MaxString;
	(* TwinCAT printf with the test message *)
	messageStringBuilder	:Tc2_Utilities.FB_FormatString;
END_VAR
THIS^.assertorContainer.resetAssertor();

assertionIsWrong := (valueToTest > maximum);
message := SEL(
	assertionIsWrong,
	'currentValue is %d maximumValue is %d assertion must be TRUE',
	'currentValue is %d maximumValue is %d assertion must be FALSE'
);
messageStringBuilder(
	sFormat := message,
	arg1 := THIS^.AnyToArg(valueToTest),
	arg2 := THIS^.AnyToArg(maximum)
);

THIS^.assertorContainer.assertor.assert.bitNumber.long.valueIsMax(
	currentValue := valueToTest,
	maximumValue := maximum,
	message := ''
);

THIS^.AssertEquals_BOOL(
	Expected 	:= assertionIsWrong,
	Actual 		:= THIS^.assertorContainer.wasAssertionWrong,
	Message 	:= messageStringBuilder.sOut
);
END_METHOD

(*

long summary
==================
This test method tests ``assert.bitNumber.long.valueIsMin``
method of CNM_AssertionInterfaces library, 
it provides the possibility to handover test data via parameter 


.. <legal notes>

legal notes
=================
| SPDX-FileCopyrightText: © 2022 ekvip automation GmbH <info@ekvip.de>
| SPDX-License-Identifier: Apache-2.0
| For details check: Apache-2.0_

.. _Apache-2.0: https://www.apache.org/licenses/LICENSE-2.0

.. </legal notes>

parameters
==========

*)

METHOD testValueIsMin 
VAR_INPUT
	(* for the test it's the parameter ``currentValue`` *)
	valueToTest	:LWORD;
	(* for the test it's the parameter ``minimumValue`` *)
	minimum		:LWORD;
END_VAR
VAR
	(* just the expectation if the assertion to test must be worng or true *)
	assertionIsWrong		:BOOL;
	(* contains the format string for the test message *)
	message					:Tc2_System.T_MaxString;
	(* TwinCAT printf with the test message *)
	messageStringBuilder	:Tc2_Utilities.FB_FormatString;
END_VAR
THIS^.assertorContainer.resetAssertor();

assertionIsWrong := (valueToTest < minimum);
message := SEL(
	assertionIsWrong,
	'currentValue is %d minimumValue is %d assertion must be TRUE',
	'currentValue is %d minimumValue is %d assertion must be FALSE'
);
messageStringBuilder(
	sFormat := message,
	arg1 := THIS^.AnyToArg(valueToTest),
	arg2 := THIS^.AnyToArg(minimum)
);

THIS^.assertorContainer.assertor.assert.bitNumber.long.valueIsMin(
	currentValue := valueToTest,
	minimumValue := minimum,
	message := ''
);

THIS^.AssertEquals_BOOL(
	Expected 	:= assertionIsWrong,
	Actual 		:= THIS^.assertorContainer.wasAssertionWrong,
	Message 	:= messageStringBuilder.sOut
);
END_METHOD

(*

long summary
==================
This test method tests ``assert.bitNumber.long.valueIsNotEqualTo``
method of CNM_AssertionInterfaces library, 
it provides the possibility to handover test data via parameter 


.. <legal notes>

legal notes
=================
| SPDX-FileCopyrightText: © 2022 ekvip automation GmbH <info@ekvip.de>
| SPDX-License-Identifier: Apache-2.0
| For details check: Apache-2.0_

.. _Apache-2.0: https://www.apache.org/licenses/LICENSE-2.0

.. </legal notes>

parameters
==========

*)

METHOD testValueIsNotEqualTo
VAR_INPUT
	(* for the test it's the parameter ``currentValue`` *)
	valueToTest	:LWORD;
	(* for the test it's the parameter ``unexpectedValue`` *)
	unexpected	:LWORD;
END_VAR
VAR
	(* just the expectation if the assertion to test must be worng or true *)
	assertionIsWrong		:BOOL;
	(* contains the format string for the test message *)
	message					:Tc2_System.T_MaxString;
	(* TwinCAT printf with the test message *)
	messageStringBuilder	:Tc2_Utilities.FB_FormatString;
END_VAR
THIS^.assertorContainer.resetAssertor();

assertionIsWrong := (valueToTest = unexpected);
message := SEL(
	assertionIsWrong,
	'currentValue is %d unexpectedValue is %d assertion must be TRUE', 
	'currentValue is %d unexpectedValue is %d assertion must be FALSE'
);
messageStringBuilder(
	sFormat := message,
	arg1 := THIS^.AnyToArg(valueToTest),
	arg2 := THIS^.AnyToArg(unexpected)
);

THIS^.assertorContainer.assertor.assert.bitNumber.long.valueIsNotEqualTo(
	currentValue := valueToTest,
	unexpectedValue := unexpected,
	message := ''
);

THIS^.AssertEquals_BOOL(
	Expected 	:= assertionIsWrong,
	Actual 		:= THIS^.assertorContainer.wasAssertionWrong,
	Message 	:= messageStringBuilder.sOut
);
END_METHOD

(*

long summary
==================
This test method tests ``assert.bitNumber.long.xorMaskIsEqualTo``
method of CNM_AssertionInterfaces library, 
it provides the possibility to handover test data via parameter 


.. <legal notes>

legal notes
=================
| SPDX-FileCopyrightText: © 2022 ekvip automation GmbH <info@ekvip.de>
| SPDX-License-Identifier: Apache-2.0
| For details check: Apache-2.0_

.. _Apache-2.0: https://www.apache.org/licenses/LICENSE-2.0

.. </legal notes>

parameters
==========

*)

METHOD testXorMaskIsEqualTo 
VAR_INPUT
	(* for the test it's the parameter ``currentValue`` *)
	valueToTest	:LWORD;
	(* it's the mask for the currentValue *)
	mask		:LWORD;
	(* for the test it's the parameter ``expectedValue`` *)
	expected	:LWORD;
END_VAR
VAR
	(* just the expectation if the assertion to test must be worng or true *)
	assertionIsWrong		:BOOL;
	(* result of the bit operation to determine the value of ``assertionIsWrong`` *)
	result					:LWORD;
	(* contains the format string for the test message *)
	message					:Tc2_System.T_MaxString;
	(* TwinCAT printf with the test message *)
	messageStringBuilder	:Tc2_Utilities.FB_FormatString;
END_VAR
THIS^.assertorContainer.resetAssertor();

result := (valueToTest XOR mask);
assertionIsWrong := (result <> expected);
message := SEL(
	assertionIsWrong,
	'currentValue: 16#%.16X XOR mask: 16#%.16X is 16#%.16X expectedValue: 16#%.16X assertion must be TRUE', 
	'currentValue: 16#%.16X XOR mask: 16#%.16X is 16#%.16X expectedValue: 16#%.16X assertion must be FALSE'
);
messageStringBuilder(
	sFormat := message,
	arg1 := THIS^.AnyToArg(valueToTest),
	arg2 := THIS^.AnyToArg(mask),
	arg3 := THIS^.AnyToArg(result),
	arg4 := THIS^.AnyToArg(expected)
);

THIS^.assertorContainer.assertor.assert.bitNumber.long.xorMaskIsEqualTo(
	currentValue	:= valueToTest,
	mask 			:= mask,
	expectedValue	:= expected,
	message			:= ''
);

THIS^.AssertEquals_BOOL(
	Expected 	:= assertionIsWrong,
	Actual 		:= THIS^.assertorContainer.wasAssertionWrong,
	Message 	:= messageStringBuilder.sOut
);
END_METHOD

(*

long summary
==================
This test method tests ``assert.bitNumber.long.xorMaskIsNotEqualTo``
method of CNM_AssertionInterfaces library, 
it provides the possibility to handover test data via parameter 


.. <legal notes>

legal notes
=================
| SPDX-FileCopyrightText: © 2022 ekvip automation GmbH <info@ekvip.de>
| SPDX-License-Identifier: Apache-2.0
| For details check: Apache-2.0_

.. _Apache-2.0: https://www.apache.org/licenses/LICENSE-2.0

.. </legal notes>

parameters
==========

*)

METHOD testXorMaskIsNotEqualTo 
VAR_INPUT
	(* for the test it's the parameter ``currentValue`` *)
	valueToTest	:LWORD;
	(* it's the mask for the currentValue *)
	mask		:LWORD;
	(* for the test it's the parameter ``unexpectedValue`` *)
	unexpected	:LWORD;
END_VAR
VAR
	(* just the expectation if the assertion to test must be worng or true *)
	assertionIsWrong		:BOOL;
	(* result of the bit operation to determine the value of ``assertionIsWrong`` *)
	result					:LWORD;
	(* contains the format string for the test message *)
	message					:Tc2_System.T_MaxString;
	(* TwinCAT printf with the test message *)
	messageStringBuilder	:Tc2_Utilities.FB_FormatString;
END_VAR
THIS^.assertorContainer.resetAssertor();

result := (valueToTest XOR mask);
assertionIsWrong := (result = unexpected);
message := SEL(
	assertionIsWrong,
	'currentValue: 16#%.16X XOR mask: 16#%.16X is 16#%.16X unexpectedValue: 16#%.16X assertion must be TRUE', 
	'currentValue: 16#%.16X XOR mask: 16#%.16X is 16#%.16X unexpectedValue: 16#%.16X assertion must be FALSE'
);
messageStringBuilder(
	sFormat := message,
	arg1 := THIS^.AnyToArg(valueToTest),
	arg2 := THIS^.AnyToArg(mask),
	arg3 := THIS^.AnyToArg(result),
	arg4 := THIS^.AnyToArg(unexpected)
);

THIS^.assertorContainer.assertor.assert.bitNumber.long.xorMaskIsNotEqualTo(
	currentValue	:= valueToTest,
	mask 			:= mask,
	unexpectedValue	:= unexpected,
	message			:= ''
);

THIS^.AssertEquals_BOOL(
	Expected 	:= assertionIsWrong,
	Actual 		:= THIS^.assertorContainer.wasAssertionWrong,
	Message 	:= messageStringBuilder.sOut
);
END_METHOD

END_FUNCTION_BLOCK

// ---- AssertionTester/AssertionTests/BitNumberAssertions/classes/DWordAssertionTests.TcPOU
(*

double summary
==================
This class tests all methods of DWORD assertions
with various combinations of inputs and checks expected 
outputs are satisfied or not

.. <legal notes>

legal notes
=================
| SPDX-FileCopyrightText: © 2022 ekvip automation GmbH <info@ekvip.de>
| SPDX-License-Identifier: Apache-2.0
| For details check: Apache-2.0_

.. _Apache-2.0: https://www.apache.org/licenses/LICENSE-2.0

.. </legal notes>

methods and properties
======================

*)

FUNCTION_BLOCK DWordAssertionTests EXTENDS AbstractAssertorTest
VAR_INPUT
END_VAR
VAR CONSTANT
	(* number of the lsb *)
	FIRST_BIT				:USINT := 0;
	(* number of the msb *)
	LAST_BIT				:USINT := 31;
	(* just the value zero *)
	ZERO					:DINT := 0;
	(* no single bit is set, it's just the value zero *)
	NO_BIT_SET				:DWORD := 16#0000_0000;
	(* just the lsb is set, it's just the value one *)
	LSB_ONLY				:DWORD := 16#0000_0001;
	(* all bits are set *)
	ALL_BITS_SET			:DWORD := 16#FFFF_FFFF;
	(* the msb is set only *)
	MSB_ONLY				:DWORD := 16#8000_0000;
	(* prefix to unify the test names *)
	TEST_NAME_PREFIX		:STRING := 'assert.bitNumber.double.';
	(* number how many times the product will be rotated right *)
	NUMBER_OF_RORS			:UDINT := 1;
	(* multiplicand for the ``multiplier`` *)
	MULTIPLICAND			:UDINT := 16#1111_1111;
	(* first of all multipliers the test iterates *)
	FIRST_MULTIPLIER		:UDINT := 0;
	(* first of all multipliers the test iterates *)
	LAST_MULTIPLIER			:UDINT := 15;
	(* constant for the modulo operator to check if valueToTest is even (lsb is unset) or odd (lsb is set) *)
	DEVISOR_FOR_EVEN_ODD	:UDINT := 2;
END_VAR

